LIN {X 0,Y 189.599,Z 448.711,A -85,B 0,C 180,E1 -22382.4,E2 -22382.4} C_VEL
LIN {X 0,Y 185.907,Z 453.993,A -85,B 0,C 180,E1 -22385.43,E2 -22385.43} C_VEL
LIN {X 0,Y 182.746,Z 458.185,A -85,B 0,C 180,E1 -22388.573,E2 -22388.573} C_VEL
LIN {X 0,Y 180.103,Z 461.393,A -85,B 0,C 180,E1 -22391.811,E2 -22391.811} C_VEL
LIN {X 0,Y 178.683,Z 463.032,A -85,B 0,C 180,E1 -22394.02,E2 -22394.02} C_VEL
LIN {X 0,Y 176.938,Z 465.065,A -85,B 0,C 180,E1 -22398.546,E2 -22398.546} C_VEL
LIN {X 0,Y 176.13,Z 465.589,A -85,B 0,C 180,E1 -22403.125,E2 -22403.125} C_VEL
LIN {X 0,Y 176.1,Z 465.056,A -85,B 0,C 180,E1 -22406.147,E2 -22406.147} C_VEL
LIN {X 0,Y 176.317,Z 464.526,A -85,B 0,C 180,E1 -22407.716,E2 -22407.716} C_VEL
LIN {X 0,Y 176.425,Z 463.36,A -85,B 0,C 180,E1 -22410,E2 -22410} C_VEL
LIN {X 0,Y 176.412,Z 461.752,A -85,B 0,C 180,E1 -22412.283,E2 -22412.283} C_VEL
LIN {X 0,Y 176.345,Z 458.528,A -85,B 0,C 180,E1 -22415.603,E2 -22415.603} C_VEL
LIN {X 0,Y 176.58,Z 453.896,A -85,B 0,C 180,E1 -22419.159,E2 -22419.159} C_VEL
LIN {X 0,Y 177.26,Z 448.101,A -85,B 0,C 180,E1 -22422.594,E2 -22422.594} C_VEL
LIN {X 0,Y 178.483,Z 440.77,A -85,B 0,C 180,E1 -22425.998,E2 -22425.998} C_VEL
LIN {X 0,Y 179.896,Z 433.284,A -85,B 0,C 180,E1 -22428.8,E2 -22428.8} C_VEL
LIN {X 0,Y 181.89,Z 423.485,A -85,B 0,C 180,E1 -22431.754,E2 -22431.754} C_VEL
LIN {X 0,Y 183.937,Z 412.997,A -85,B 0,C 180,E1 -22434.248,E2 -22434.248} C_VEL
LIN {X 0,Y 186.015,Z 401.711,A -85,B 0,C 180,E1 -22436.352,E2 -22436.352} C_VEL
LIN {X 0,Y 188.191,Z 389.227,A -85,B 0,C 180,E1 -22438.127,E2 -22438.127} C_VEL
LIN {X 0,Y 189.916,Z 375.866,A -85,B 0,C 180,E1 -22439.51,E2 -22439.51} C_VEL
LIN {X 0,Y 191.178,Z 362.832,A -85,B 0,C 180,E1 -22440.435,E2 -22440.435} C_VEL
LIN {X 0,Y 193.662,Z 313.849,A -85,B 0,C 180,E1 -22442.625,E2 -22442.625} C_VEL
LIN {X 0,Y 190.578,Z 284.083,A -85,B 0,C 180,E1 -22444.515,E2 -22444.515} C_VEL
LIN {X 0,Y 182.555,Z 261.017,A -85,B 0,C 180,E1 -22446.816,E2 -22446.816} C_VEL
LIN {X 0,Y 180.086,Z 254.3,A -85,B 0,C 180,E1 -22447.559,E2 -22447.559} C_VEL
LIN {X 0,Y 178.442,Z 247.259,A -85,B 0,C 180,E1 -22451.351,E2 -22451.351} C_VEL
LIN {X 0,Y 178.382,Z 247.27,A -85,B 0,C 180,E1 -22455.161,E2 -22455.161} C_VEL
LIN {X 0,Y 178.388,Z 247.265,A -85,B 0,C 180,E1 -22458.457,E2 -22458.457} C_VEL
LIN {X 0,Y 178.406,Z 247.261,A -85,B 0,C 180,E1 -22463.778,E2 -22463.778} C_VEL
LIN {X 0,Y 178.468,Z 247.249,A -85,B 0,C 180,E1 -22466.542,E2 -22466.542} C_VEL
LIN {X 0,Y 178.434,Z 247.254,A -85,B 0,C 180,E1 -22471.793,E2 -22471.793} C_VEL
LIN {X 0,Y 178.5,Z 247.242,A -85,B 0,C 180,E1 -22474.886,E2 -22474.886} C_VEL
LIN {X 0,Y 178.587,Z 247.231,A -85,B 0,C 180,E1 -22481.649,E2 -22481.649} C_VEL
LIN {X 0,Y 178.618,Z 247.225,A -85,B 0,C 180,E1 -22486.344,E2 -22486.344} C_VEL
LIN {X 0,Y 178.883,Z 247.204,A -85,B 0,C 180,E1 -22490.958,E2 -22490.958} C_VEL
LIN {X 0,Y 179.11,Z 247.151,A -85,B 0,C 180,E1 -22497.75,E2 -22497.75} C_VEL
LIN {X 0,Y 179.333,Z 247.119,A -85,B 0,C 180,E1 -22499.999,E2 -22499.999} C_VEL
LIN {X 0,Y 178.829,Z 247.202,A -85,B 0,C 180,E1 -22504.507,E2 -22504.507} C_VEL
LIN {X 0,Y 178.883,Z 247.202,A -85,B 0,C 180,E1 -22509.041,E2 -22509.041} C_VEL
LIN {X 0,Y 178.629,Z 247.222,A -85,B 0,C 180,E1 -22513.654,E2 -22513.654} C_VEL
LIN {X 0,Y 178.635,Z 247.195,A -85,B 0,C 180,E1 -22519.245,E2 -22519.245} C_VEL
LIN {X 0,Y 178.517,Z 247.242,A -85,B 0,C 180,E1 -22525.126,E2 -22525.126} C_VEL
LIN {X 0,Y 178.505,Z 247.249,A -85,B 0,C 180,E1 -22529.995,E2 -22529.995} C_VEL
LIN {X 0,Y 178.474,Z 247.243,A -85,B 0,C 180,E1 -22534.224,E2 -22534.224} C_VEL
LIN {X 0,Y 178.431,Z 247.223,A -85,B 0,C 180,E1 -22539.064,E2 -22539.064} C_VEL
LIN {X 0,Y 178.432,Z 247.234,A -85,B 0,C 180,E1 -22542.034,E2 -22542.034} C_VEL
LIN {X 0,Y 178.414,Z 247.253,A -85,B 0,C 180,E1 -22545.156,E2 -22545.156} C_VEL
LIN {X 0,Y 178.397,Z 247.263,A -85,B 0,C 180,E1 -22548.46,E2 -22548.46} C_VEL
LIN {X 0,Y 178.412,Z 247.252,A -85,B 0,C 180,E1 -22553.786,E2 -22553.786} C_VEL
LIN {X 0,Y 178.477,Z 247.23,A -85,B 0,C 180,E1 -22556.549,E2 -22556.549} C_VEL
LIN {X 0,Y 178.515,Z 247.234,A -85,B 0,C 180,E1 -22560.01,E2 -22560.01} C_VEL
LIN {X 0,Y 178.529,Z 247.246,A -85,B 0,C 180,E1 -22564.878,E2 -22564.878} C_VEL
LIN {X 0,Y 178.619,Z 247.221,A -85,B 0,C 180,E1 -22570.786,E2 -22570.786} C_VEL
LIN {X 0,Y 178.662,Z 247.228,A -85,B 0,C 180,E1 -22574.019,E2 -22574.019} C_VEL
LIN {X 0,Y 178.859,Z 247.2,A -85,B 0,C 180,E1 -22579.211,E2 -22579.211} C_VEL
LIN {X 0,Y 178.923,Z 247.198,A -85,B 0,C 180,E1 -22583.234,E2 -22583.234} C_VEL
LIN {X 0,Y 179.152,Z 247.165,A -85,B 0,C 180,E1 -22587.752,E2 -22587.752} C_VEL
LIN {X 0,Y 179.369,Z 247.142,A -85,B 0,C 180,E1 -22590,E2 -22590} C_VEL
LIN {X 0,Y 178.869,Z 247.204,A -85,B 0,C 180,E1 -22594.507,E2 -22594.507} C_VEL
LIN {X 0,Y 178.922,Z 247.2,A -85,B 0,C 180,E1 -22599.039,E2 -22599.039} C_VEL
LIN {X 0,Y 178.707,Z 247.228,A -85,B 0,C 180,E1 -22602.793,E2 -22602.793} C_VEL
LIN {X 0,Y 179.772,Z 250.154,A -85,B 0,C 180,E1 -22603.121,E2 -22603.121} C_VEL
LIN {X 0,Y 187.477,Z 267.491,A -85,B 0,C 180,E1 -22605.177,E2 -22605.177} C_VEL
LIN {X 0,Y 194.565,Z 285.188,A -85,B 0,C 180,E1 -22606.986,E2 -22606.986} C_VEL
LIN {X 0,Y 194.878,Z 286.201,A -85,B 0,C 180,E1 -22607.076,E2 -22607.076} C_VEL
LIN {X 0,Y 191.309,Z 347.18,A -85,B 0,C 180,E1 -22609.758,E2 -22609.758} C_VEL
LIN {X 0,Y 190.227,Z 360,A -85,B 0,C 180,E1 -22610.722,E2 -22610.722} C_VEL
LIN {X 0,Y 188.85,Z 371.973,A -85,B 0,C 180,E1 -22611.989,E2 -22611.989} C_VEL
LIN {X 0,Y 186.955,Z 384.854,A -85,B 0,C 180,E1 -22613.833,E2 -22613.833} C_VEL
LIN {X 0,Y 184.919,Z 396.527,A -85,B 0,C 180,E1 -22616.003,E2 -22616.003} C_VEL
LIN {X 0,Y 182.877,Z 407.104,A -85,B 0,C 180,E1 -22618.514,E2 -22618.514} C_VEL
LIN {X 0,Y 181.019,Z 416.582,A -85,B 0,C 180,E1 -22621.337,E2 -22621.337} C_VEL
LIN {X 0,Y 179.188,Z 425.253,A -85,B 0,C 180,E1 -22624.55,E2 -22624.55} C_VEL
LIN {X 0,Y 177.846,Z 432.169,A -85,B 0,C 180,E1 -22627.783,E2 -22627.783} C_VEL
LIN {X 0,Y 176.977,Z 437.712,A -85,B 0,C 180,E1 -22631.018,E2 -22631.018} C_VEL
LIN {X 0,Y 176.14,Z 443.11,A -85,B 0,C 180,E1 -22635.12,E2 -22635.12} C_VEL
LIN {X 0,Y 175.887,Z 445.264,A -85,B 0,C 180,E1 -22637.214,E2 -22637.214} C_VEL
LIN {X 0,Y 175.78,Z 447.658,A -85,B 0,C 180,E1 -22640.231,E2 -22640.231} C_VEL
LIN {X 0,Y 175.992,Z 449.322,A -85,B 0,C 180,E1 -22643.202,E2 -22643.202} C_VEL
LIN {X 0,Y 176.702,Z 450.396,A -85,B 0,C 180,E1 -22646.631,E2 -22646.631} C_VEL
LIN {X 0,Y 177.97,Z 450.542,A -85,B 0,C 180,E1 -22650.306,E2 -22650.306} C_VEL
LIN {X 0,Y 180.201,Z 449.345,A -85,B 0,C 180,E1 -22654.596,E2 -22654.596} C_VEL
LIN {X 0,Y 182.337,Z 447.564,A -85,B 0,C 180,E1 -22657.662,E2 -22657.662} C_VEL
LIN {X 0,Y 185.512,Z 444.303,A -85,B 0,C 180,E1 -22661.264,E2 -22661.264} C_VEL
LIN {X 0,Y 189.738,Z 439.371,A -85,B 0,C 180,E1 -22664.973,E2 -22664.973} C_VEL
LIN {X 0,Y 193.955,Z 433.791,A -85,B 0,C 180,E1 -22668.027,E2 -22668.027} C_VEL
LIN {X 0,Y 197.968,Z 427.738,A -85,B 0,C 180,E1 -22670.602,E2 -22670.602} C_VEL
LIN {X 0,Y 202.399,Z 420.472,A -85,B 0,C 180,E1 -22673.02,E2 -22673.02} C_VEL
LIN {X 0,Y 207.339,Z 411.368,A -85,B 0,C 180,E1 -22675.383,E2 -22675.383} C_VEL
LIN {X 0,Y 212.434,Z 400.451,A -85,B 0,C 180,E1 -22677.574,E2 -22677.574} C_VEL
LIN {X 0,Y 216.736,Z 389.318,A -85,B 0,C 180,E1 -22679.289,E2 -22679.289} C_VEL
LIN {X 0,Y 220.567,Z 377.326,A -85,B 0,C 180,E1 -22680.685,E2 -22680.685} C_VEL
LIN {X 0,Y 223.601,Z 364.833,A -85,B 0,C 180,E1 -22681.802,E2 -22681.802} C_VEL
LIN {X 0,Y 225.801,Z 352.533,A -85,B 0,C 180,E1 -22682.584,E2 -22682.584} C_VEL
LIN {X 0,Y 228.467,Z 329.492,A -85,B 0,C 180,E1 -22683.486,E2 -22683.486} C_VEL
LIN {X 0,Y 230.182,Z 313.067,A -85,B 0,C 180,E1 -22684.103,E2 -22684.103} C_VEL
LIN {X 0,Y 226.331,Z 304.592,A -85,B 0,C 180,E1 -22686.72,E2 -22686.72} C_VEL
LIN {X 0,Y 224.187,Z 300.987,A -85,B 0,C 180,E1 -22688.303,E2 -22688.303} C_VEL
LIN {X 0,Y 221.023,Z 295.846,A -85,B 0,C 180,E1 -22690.999,E2 -22690.999} C_VEL
LIN {X 0,Y 219.416,Z 293.216,A -85,B 0,C 180,E1 -22692.625,E2 -22692.625} C_VEL
LIN {X 0,Y 217.287,Z 290.254,A -85,B 0,C 180,E1 -22695.197,E2 -22695.197} C_VEL
LIN {X 0,Y 215.463,Z 287.989,A -85,B 0,C 180,E1 -22698.105,E2 -22698.105} C_VEL
LIN {X 0,Y 214.273,Z 286.482,A -85,B 0,C 180,E1 -22701.15,E2 -22701.15} C_VEL
LIN {X 0,Y 213.854,Z 286.773,A -85,B 0,C 180,E1 -22706.485,E2 -22706.485} C_VEL
LIN {X 0,Y 214.9,Z 288.985,A -85,B 0,C 180,E1 -22710.453,E2 -22710.453} C_VEL
LIN {X 0,Y 217.907,Z 295.087,A -85,B 0,C 180,E1 -22715.571,E2 -22715.571} C_VEL
LIN {X 0,Y 220.497,Z 300.345,A -85,B 0,C 180,E1 -22718.445,E2 -22718.445} C_VEL
LIN {X 0,Y 223.12,Z 306.049,A -85,B 0,C 180,E1 -22720.845,E2 -22720.845} C_VEL
LIN {X 0,Y 225.734,Z 312.199,A -85,B 0,C 180,E1 -22722.959,E2 -22722.959} C_VEL
LIN {X 0,Y 228.58,Z 319.942,A -85,B 0,C 180,E1 -22725.006,E2 -22725.006} C_VEL
LIN {X 0,Y 229.366,Z 322.663,A -85,B 0,C 180,E1 -22725.588,E2 -22725.588} C_VEL
LIN {X 0,Y 229.11,Z 326.685,A -85,B 0,C 180,E1 -22725.81,E2 -22725.81} C_VEL
LIN {X 0,Y 225.297,Z 360.929,A -85,B 0,C 180,E1 -22727.075,E2 -22727.075} C_VEL
LIN {X 0,Y 224.524,Z 365.452,A -85,B 0,C 180,E1 -22727.265,E2 -22727.265} C_VEL
LIN {X 0,Y 223.429,Z 369.295,A -85,B 0,C 180,E1 -22727.323,E2 -22727.323} C_VEL
LIN {X 0,Y 217.491,Z 381.326,A -85,B 0,C 180,E1 -22726.845,E2 -22726.845} C_VEL
LIN {X 0,Y 216.118,Z 384.997,A -85,B 0,C 180,E1 -22727.019,E2 -22727.019} C_VEL
LIN {X 0,Y 212.124,Z 396.806,A -85,B 0,C 180,E1 -22728.187,E2 -22728.187} C_VEL
LIN {X 0,Y 207.021,Z 409.179,A -85,B 0,C 180,E1 -22729.838,E2 -22729.838} C_VEL
LIN {X 0,Y 201.733,Z 420.185,A -85,B 0,C 180,E1 -22731.807,E2 -22731.807} C_VEL
LIN {X 0,Y 196.789,Z 429.15,A -85,B 0,C 180,E1 -22733.899,E2 -22733.899} C_VEL
LIN {X 0,Y 191.316,Z 437.995,A -85,B 0,C 180,E1 -22736.567,E2 -22736.567} C_VEL
LIN {X 0,Y 186.364,Z 445.214,A -85,B 0,C 180,E1 -22739.4,E2 -22739.4} C_VEL
LIN {X 0,Y 181.983,Z 451.123,A -85,B 0,C 180,E1 -22742.395,E2 -22742.395} C_VEL
LIN {X 0,Y 178.293,Z 455.843,A -85,B 0,C 180,E1 -22745.553,E2 -22745.553} C_VEL
LIN {X 0,Y 175.164,Z 459.516,A -85,B 0,C 180,E1 -22748.834,E2 -22748.834} C_VEL
LIN {X 0,Y 173.364,Z 461.453,A -85,B 0,C 180,E1 -22751.078,E2 -22751.078} C_VEL
LIN {X 0,Y 170.739,Z 464.082,A -85,B 0,C 180,E1 -22755.703,E2 -22755.703} C_VEL
LIN {X 0,Y 169.386,Z 465.213,A -85,B 0,C 180,E1 -22760.448,E2 -22760.448} C_VEL
LIN {X 0,Y 169.082,Z 465.187,A -85,B 0,C 180,E1 -22762.837,E2 -22762.837} C_VEL
LIN {X 0,Y 169.242,Z 463.955,A -85,B 0,C 180,E1 -22767.62,E2 -22767.62} C_VEL
LIN {X 0,Y 169.364,Z 462.725,A -85,B 0,C 180,E1 -22770,E2 -22770} C_VEL
LIN {X 0,Y 169.269,Z 459.946,A -85,B 0,C 180,E1 -22773.591,E2 -22773.591} C_VEL
LIN {X 0,Y 169.327,Z 456.088,A -85,B 0,C 180,E1 -22777.152,E2 -22777.152} C_VEL
LIN {X 0,Y 169.771,Z 451,A -85,B 0,C 180,E1 -22780.735,E2 -22780.735} C_VEL
LIN {X 0,Y 170.659,Z 444.517,A -85,B 0,C 180,E1 -22784.303,E2 -22784.303} C_VEL
LIN {X 0,Y 172.216,Z 436.375,A -85,B 0,C 180,E1 -22787.82,E2 -22787.82} C_VEL
LIN {X 0,Y 173.845,Z 428.029,A -85,B 0,C 180,E1 -22790.713,E2 -22790.713} C_VEL
LIN {X 0,Y 175.971,Z 417.858,A -85,B 0,C 180,E1 -22793.537,E2 -22793.537} C_VEL
LIN {X 0,Y 178.275,Z 406.408,A -85,B 0,C 180,E1 -22796.01,E2 -22796.01} C_VEL
LIN {X 0,Y 180.296,Z 395.287,A -85,B 0,C 180,E1 -22797.886,E2 -22797.886} C_VEL
LIN {X 0,Y 182.206,Z 383.022,A -85,B 0,C 180,E1 -22799.454,E2 -22799.454} C_VEL
LIN {X 0,Y 183.801,Z 369.682,A -85,B 0,C 180,E1 -22800.675,E2 -22800.675} C_VEL
LIN {X 0,Y 184.836,Z 356.969,A -85,B 0,C 180,E1 -22801.437,E2 -22801.437} C_VEL
LIN {X 0,Y 187.018,Z 314.116,A -85,B 0,C 180,E1 -22803.404,E2 -22803.404} C_VEL
LIN {X 0,Y 184.2,Z 286.195,A -85,B 0,C 180,E1 -22805.224,E2 -22805.224} C_VEL
LIN {X 0,Y 176.567,Z 264.085,A -85,B 0,C 180,E1 -22807.542,E2 -22807.542} C_VEL
LIN {X 0,Y 172.741,Z 253.927,A -85,B 0,C 180,E1 -22808.734,E2 -22808.734} C_VEL
LIN {X 0,Y 171.377,Z 248.14,A -85,B 0,C 180,E1 -22812,E2 -22812} C_VEL
LIN {X 0,Y 171.322,Z 248.148,A -85,B 0,C 180,E1 -22817.588,E2 -22817.588} C_VEL
LIN {X 0,Y 171.348,Z 248.142,A -85,B 0,C 180,E1 -22822.03,E2 -22822.03} C_VEL
LIN {X 0,Y 171.385,Z 248.132,A -85,B 0,C 180,E1 -22825.09,E2 -22825.09} C_VEL
LIN {X 0,Y 171.397,Z 248.135,A -85,B 0,C 180,E1 -22830.524,E2 -22830.524} C_VEL
LIN {X 0,Y 171.419,Z 248.129,A -85,B 0,C 180,E1 -22835.795,E2 -22835.795} C_VEL
LIN {X 0,Y 171.488,Z 248.12,A -85,B 0,C 180,E1 -22840.86,E2 -22840.86} C_VEL
LIN {X 0,Y 171.533,Z 248.105,A -85,B 0,C 180,E1 -22845.768,E2 -22845.768} C_VEL
LIN {X 0,Y 171.822,Z 248.082,A -85,B 0,C 180,E1 -22850.583,E2 -22850.583} C_VEL
LIN {X 0,Y 171.774,Z 248.076,A -85,B 0,C 180,E1 -22855.305,E2 -22855.305} C_VEL
LIN {X 0,Y 172.297,Z 247.994,A -85,B 0,C 180,E1 -22859.999,E2 -22859.999} C_VEL
LIN {X 0,Y 171.778,Z 248.081,A -85,B 0,C 180,E1 -22864.693,E2 -22864.693} C_VEL
LIN {X 0,Y 171.822,Z 248.08,A -85,B 0,C 180,E1 -22869.416,E2 -22869.416} C_VEL
LIN {X 0,Y 171.549,Z 248.1,A -85,B 0,C 180,E1 -22874.229,E2 -22874.229} C_VEL
LIN {X 0,Y 171.557,Z 248.077,A -85,B 0,C 180,E1 -22879.591,E2 -22879.591} C_VEL
LIN {X 0,Y 171.452,Z 248.121,A -85,B 0,C 180,E1 -22885.617,E2 -22885.617} C_VEL
LIN {X 0,Y 171.423,Z 248.131,A -85,B 0,C 180,E1 -22890.587,E2 -22890.587} C_VEL
LIN {X 0,Y 171.386,Z 248.122,A -85,B 0,C 180,E1 -22895.035,E2 -22895.035} C_VEL
LIN {X 0,Y 171.387,Z 248.099,A -85,B 0,C 180,E1 -22898.828,E2 -22898.828} C_VEL
LIN {X 0,Y 171.342,Z 248.129,A -85,B 0,C 180,E1 -22904.209,E2 -22904.209} C_VEL
LIN {X 0,Y 171.328,Z 248.142,A -85,B 0,C 180,E1 -22908.985,E2 -22908.985} C_VEL
LIN {X 0,Y 171.376,Z 248.134,A -85,B 0,C 180,E1 -22912.043,E2 -22912.043} C_VEL
LIN {X 0,Y 171.389,Z 248.121,A -85,B 0,C 180,E1 -22915.095,E2 -22915.095} C_VEL
LIN {X 0,Y 171.442,Z 248.119,A -85,B 0,C 180,E1 -22920.537,E2 -22920.537} C_VEL
LIN {X 0,Y 171.453,Z 248.129,A -85,B 0,C 180,E1 -22925.804,E2 -22925.804} C_VEL
LIN {X 0,Y 171.575,Z 248.097,A -85,B 0,C 180,E1 -22930.874,E2 -22930.874} C_VEL
LIN {X 0,Y 171.607,Z 248.11,A -85,B 0,C 180,E1 -22935.777,E2 -22935.777} C_VEL
LIN {X 0,Y 171.871,Z 248.065,A -85,B 0,C 180,E1 -22940.587,E2 -22940.587} C_VEL
LIN {X 0,Y 171.821,Z 248.084,A -85,B 0,C 180,E1 -22945.308,E2 -22945.308} C_VEL
LIN {X 0,Y 172.332,Z 248.019,A -85,B 0,C 180,E1 -22950,E2 -22950} C_VEL
LIN {X 0,Y 171.818,Z 248.083,A -85,B 0,C 180,E1 -22954.692,E2 -22954.692} C_VEL
LIN {X 0,Y 171.86,Z 248.079,A -85,B 0,C 180,E1 -22959.414,E2 -22959.414} C_VEL
LIN {X 0,Y 171.734,Z 248.097,A -85,B 0,C 180,E1 -22961.7,E2 -22961.7} C_VEL
LIN {X 0,Y 172.764,Z 251.05,A -85,B 0,C 180,E1 -22962.069,E2 -22962.069} C_VEL
LIN {X 0,Y 180.588,Z 268.538,A -85,B 0,C 180,E1 -22964.262,E2 -22964.262} C_VEL
LIN {X 0,Y 188.151,Z 287.318,A -85,B 0,C 180,E1 -22966.296,E2 -22966.296} C_VEL
LIN {X 0,Y 184.635,Z 347.103,A -85,B 0,C 180,E1 -22969.032,E2 -22969.032} C_VEL
LIN {X 0,Y 183.493,Z 360.308,A -85,B 0,C 180,E1 -22970.053,E2 -22970.053} C_VEL
LIN {X 0,Y 182.053,Z 372.503,A -85,B 0,C 180,E1 -22971.391,E2 -22971.391} C_VEL
LIN {X 0,Y 180.105,Z 385.172,A -85,B 0,C 180,E1 -22973.269,E2 -22973.269} C_VEL
LIN {X 0,Y 177.949,Z 397.03,A -85,B 0,C 180,E1 -22975.553,E2 -22975.553} C_VEL
LIN {X 0,Y 175.828,Z 407.778,A -85,B 0,C 180,E1 -22978.219,E2 -22978.219} C_VEL
LIN {X 0,Y 173.75,Z 417.822,A -85,B 0,C 180,E1 -22981.359,E2 -22981.359} C_VEL
LIN {X 0,Y 171.872,Z 426.748,A -85,B 0,C 180,E1 -22984.919,E2 -22984.919} C_VEL
LIN {X 0,Y 170.5,Z 433.74,A -85,B 0,C 180,E1 -22988.449,E2 -22988.449} C_VEL
LIN {X 0,Y 169.676,Z 439.007,A -85,B 0,C 180,E1 -22991.794,E2 -22991.794} C_VEL
LIN {X 0,Y 169.046,Z 443.038,A -85,B 0,C 180,E1 -22995.029,E2 -22995.029} C_VEL
LIN {X 0,Y 168.689,Z 446.419,A -85,B 0,C 180,E1 -22998.577,E2 -22998.577} C_VEL
LIN {X 0,Y 168.802,Z 448.905,A -85,B 0,C 180,E1 -23002.277,E2 -23002.277} C_VEL
LIN {X 0,Y 169.436,Z 450.426,A -85,B 0,C 180,E1 -23006.046,E2 -23006.046} C_VEL
LIN {X 0,Y 170.875,Z 450.942,A -85,B 0,C 180,E1 -23010.427,E2 -23010.427} C_VEL
LIN {X 0,Y 172.462,Z 450.43,A -85,B 0,C 180,E1 -23013.692,E2 -23013.692} C_VEL
LIN {X 0,Y 174.948,Z 448.818,A -85,B 0,C 180,E1 -23017.497,E2 -23017.497} C_VEL
LIN {X 0,Y 178.538,Z 445.664,A -85,B 0,C 180,E1 -23021.645,E2 -23021.645} C_VEL
LIN {X 0,Y 183.291,Z 440.631,A -85,B 0,C 180,E1 -23025.805,E2 -23025.805} C_VEL
LIN {X 0,Y 188.158,Z 434.69,A -85,B 0,C 180,E1 -23029.237,E2 -23029.237} C_VEL
LIN {X 0,Y 192.925,Z 428.065,A -85,B 0,C 180,E1 -23032.149,E2 -23032.149} C_VEL
LIN {X 0,Y 198.15,Z 419.954,A -85,B 0,C 180,E1 -23034.828,E2 -23034.828} C_VEL
LIN {X 0,Y 202.612,Z 412.123,A -85,B 0,C 180,E1 -23036.854,E2 -23036.854} C_VEL
LIN {X 0,Y 207.866,Z 401.396,A -85,B 0,C 180,E1 -23039.032,E2 -23039.032} C_VEL
LIN {X 0,Y 212.257,Z 390.85,A -85,B 0,C 180,E1 -23040.697,E2 -23040.697} C_VEL
LIN {X 0,Y 216.042,Z 379.905,A -85,B 0,C 180,E1 -23042.022,E2 -23042.022} C_VEL
LIN {X 0,Y 219.409,Z 367.366,A -85,B 0,C 180,E1 -23043.204,E2 -23043.204} C_VEL
LIN {X 0,Y 221.991,Z 354.424,A -85,B 0,C 180,E1 -23044.061,E2 -23044.061} C_VEL
LIN {X 0,Y 224.248,Z 336.519,A -85,B 0,C 180,E1 -23044.797,E2 -23044.797} C_VEL
LIN {X 0,Y 226.409,Z 316.645,A -85,B 0,C 180,E1 -23045.543,E2 -23045.543} C_VEL
LIN {X 0,Y 223.518,Z 309.761,A -85,B 0,C 180,E1 -23047.766,E2 -23047.766} C_VEL
LIN {X 0,Y 220.811,Z 305.409,A -85,B 0,C 180,E1 -23049.927,E2 -23049.927} C_VEL
LIN {X 0,Y 219.147,Z 302.331,A -85,B 0,C 180,E1 -23051.555,E2 -23051.555} C_VEL
LIN {X 0,Y 217.558,Z 299.751,A -85,B 0,C 180,E1 -23053.231,E2 -23053.231} C_VEL
LIN {X 0,Y 215.64,Z 296.775,A -85,B 0,C 180,E1 -23055.79,E2 -23055.79} C_VEL
LIN {X 0,Y 214.032,Z 294.763,A -85,B 0,C 180,E1 -23058.607,E2 -23058.607} C_VEL
LIN {X 0,Y 213.075,Z 293.462,A -85,B 0,C 180,E1 -23061.274,E2 -23061.274} C_VEL
LIN {X 0,Y 212.656,Z 293.737,A -85,B 0,C 180,E1 -23066.224,E2 -23066.224} C_VEL
LIN {X 0,Y 213.536,Z 295.748,A -85,B 0,C 180,E1 -23070.011,E2 -23070.011} C_VEL
LIN {X 0,Y 216.182,Z 301.608,A -85,B 0,C 180,E1 -23074.965,E2 -23074.965} C_VEL
LIN {X 0,Y 218.488,Z 306.657,A -85,B 0,C 180,E1 -23077.761,E2 -23077.761} C_VEL
LIN {X 0,Y 220.72,Z 311.934,A -85,B 0,C 180,E1 -23080.024,E2 -23080.024} C_VEL
LIN {X 0,Y 223.064,Z 317.744,A -85,B 0,C 180,E1 -23082.045,E2 -23082.045} C_VEL
LIN {X 0,Y 225.461,Z 324.846,A -85,B 0,C 180,E1 -23083.979,E2 -23083.979} C_VEL
LIN {X 0,Y 225.706,Z 326.211,A -85,B 0,C 180,E1 -23084.217,E2 -23084.217} C_VEL
LIN {X 0,Y 221.783,Z 360.31,A -85,B 0,C 180,E1 -23085.481,E2 -23085.481} C_VEL
LIN {X 0,Y 219.295,Z 373.01,A -85,B 0,C 180,E1 -23086.135,E2 -23086.135} C_VEL
LIN {X 0,Y 216.118,Z 384.997,A -85,B 0,C 180,E1 -23087.019,E2 -23087.019} C_VEL
LIN {X 0,Y 214.102,Z 390.411,A -85,B 0,C 180,E1 -23087.386,E2 -23087.386} C_VEL
LIN {X 0,Y 209.313,Z 399.052,A -85,B 0,C 180,E1 -23087.651,E2 -23087.651} C_VEL
LIN {X 0,Y 204.132,Z 407.359,A -85,B 0,C 180,E1 -23088.068,E2 -23088.068} C_VEL
LIN {X 0,Y 201.518,Z 412.109,A -85,B 0,C 180,E1 -23088.685,E2 -23088.685} C_VEL
LIN {X 0,Y 197.401,Z 420,A -85,B 0,C 180,E1 -23090.15,E2 -23090.15} C_VEL
LIN {X 0,Y 191.188,Z 430.505,A -85,B 0,C 180,E1 -23092.665,E2 -23092.665} C_VEL
LIN {X 0,Y 185.496,Z 439.056,A -85,B 0,C 180,E1 -23095.371,E2 -23095.371} C_VEL
LIN {X 0,Y 180.338,Z 445.985,A -85,B 0,C 180,E1 -23098.261,E2 -23098.261} C_VEL
LIN {X 0,Y 174.835,Z 452.702,A -85,B 0,C 180,E1 -23102.025,E2 -23102.025} C_VEL
LIN {X 0,Y 170.672,Z 457.434,A -85,B 0,C 180,E1 -23105.686,E2 -23105.686} C_VEL
LIN {X 0,Y 168.538,Z 459.673,A -85,B 0,C 180,E1 -23107.96,E2 -23107.96} C_VEL
LIN {X 0,Y 165.046,Z 462.892,A -85,B 0,C 180,E1 -23112.66,E2 -23112.66} C_VEL
LIN {X 0,Y 162.978,Z 464.601,A -85,B 0,C 180,E1 -23117.55,E2 -23117.55} C_VEL
LIN {X 0,Y 162.017,Z 464.737,A -85,B 0,C 180,E1 -23122.523,E2 -23122.523} C_VEL
LIN {X 0,Y 162.165,Z 463.36,A -85,B 0,C 180,E1 -23127.516,E2 -23127.516} C_VEL
LIN {X 0,Y 162.304,Z 462.043,A -85,B 0,C 180,E1 -23130,E2 -23130} C_VEL
LIN {X 0,Y 162.21,Z 459.366,A -85,B 0,C 180,E1 -23133.487,E2 -23133.487} C_VEL
LIN {X 0,Y 162.267,Z 455.127,A -85,B 0,C 180,E1 -23137.465,E2 -23137.465} C_VEL
LIN {X 0,Y 162.898,Z 448.826,A -85,B 0,C 180,E1 -23141.824,E2 -23141.824} C_VEL
LIN {X 0,Y 164.014,Z 441.888,A -85,B 0,C 180,E1 -23145.532,E2 -23145.532} C_VEL
LIN {X 0,Y 165.41,Z 434.777,A -85,B 0,C 180,E1 -23148.58,E2 -23148.58} C_VEL
LIN {X 0,Y 167.192,Z 426.173,A -85,B 0,C 180,E1 -23151.578,E2 -23151.578} C_VEL
LIN {X 0,Y 169.427,Z 415.551,A -85,B 0,C 180,E1 -23154.504,E2 -23154.504} C_VEL
LIN {X 0,Y 171.586,Z 405.117,A -85,B 0,C 180,E1 -23156.775,E2 -23156.775} C_VEL
LIN {X 0,Y 173.723,Z 393.768,A -85,B 0,C 180,E1 -23158.708,E2 -23158.708} C_VEL
LIN {X 0,Y 175.694,Z 381.042,A -85,B 0,C 180,E1 -23160.329,E2 -23160.329} C_VEL
LIN {X 0,Y 177.274,Z 367.984,A -85,B 0,C 180,E1 -23161.517,E2 -23161.517} C_VEL
LIN {X 0,Y 178.305,Z 354.272,A -85,B 0,C 180,E1 -23162.311,E2 -23162.311} C_VEL
LIN {X 0,Y 180.374,Z 314.424,A -85,B 0,C 180,E1 -23164.209,E2 -23164.209} C_VEL
LIN {X 0,Y 177.684,Z 287.859,A -85,B 0,C 180,E1 -23166.035,E2 -23166.035} C_VEL
LIN {X 0,Y 170.641,Z 267.261,A -85,B 0,C 180,E1 -23168.287,E2 -23168.287} C_VEL
LIN {X 0,Y 165.369,Z 253.581,A -85,B 0,C 180,E1 -23170.011,E2 -23170.011} C_VEL
LIN {X 0,Y 164.288,Z 249.025,A -85,B 0,C 180,E1 -23172.738,E2 -23172.738} C_VEL
LIN {X 0,Y 164.251,Z 249.03,A -85,B 0,C 180,E1 -23176.794,E2 -23176.794} C_VEL
LIN {X 0,Y 164.279,Z 249.022,A -85,B 0,C 180,E1 -23180.351,E2 -23180.351} C_VEL
LIN {X 0,Y 164.313,Z 249.014,A -85,B 0,C 180,E1 -23184.348,E2 -23184.348} C_VEL
LIN {X 0,Y 164.357,Z 249.013,A -85,B 0,C 180,E1 -23189.127,E2 -23189.127} C_VEL
LIN {X 0,Y 164.38,Z 249,A -85,B 0,C 180,E1 -23194.687,E2 -23194.687} C_VEL
LIN {X 0,Y 164.4,Z 249.004,A -85,B 0,C 180,E1 -23200.115,E2 -23200.115} C_VEL
LIN {X 0,Y 164.461,Z 248.98,A -85,B 0,C 180,E1 -23205.142,E2 -23205.142} C_VEL
LIN {X 0,Y 164.744,Z 248.963,A -85,B 0,C 180,E1 -23210.174,E2 -23210.174} C_VEL
LIN {X 0,Y 164.8,Z 248.956,A -85,B 0,C 180,E1 -23212.649,E2 -23212.649} C_VEL
LIN {X 0,Y 165.261,Z 248.869,A -85,B 0,C 180,E1 -23219.999,E2 -23219.999} C_VEL
LIN {X 0,Y 164.727,Z 248.96,A -85,B 0,C 180,E1 -23224.894,E2 -23224.894} C_VEL
LIN {X 0,Y 164.801,Z 248.956,A -85,B 0,C 180,E1 -23227.349,E2 -23227.349} C_VEL
LIN {X 0,Y 164.682,Z 248.966,A -85,B 0,C 180,E1 -23231.056,E2 -23231.056} C_VEL
LIN {X 0,Y 164.478,Z 248.958,A -85,B 0,C 180,E1 -23237.403,E2 -23237.403} C_VEL
LIN {X 0,Y 164.486,Z 248.958,A -85,B 0,C 180,E1 -23239.987,E2 -23239.987} C_VEL
LIN {X 0,Y 164.376,Z 249.004,A -85,B 0,C 180,E1 -23246.135,E2 -23246.135} C_VEL
LIN {X 0,Y 164.358,Z 249.009,A -85,B 0,C 180,E1 -23251.228,E2 -23251.228} C_VEL
LIN {X 0,Y 164.301,Z 248.994,A -85,B 0,C 180,E1 -23256.787,E2 -23256.787} C_VEL
LIN {X 0,Y 164.302,Z 248.979,A -85,B 0,C 180,E1 -23259.912,E2 -23259.912} C_VEL
LIN {X 0,Y 164.295,Z 249.002,A -85,B 0,C 180,E1 -23263.355,E2 -23263.355} C_VEL
LIN {X 0,Y 164.282,Z 249.018,A -85,B 0,C 180,E1 -23266.811,E2 -23266.811} C_VEL
LIN {X 0,Y 164.286,Z 249.02,A -85,B 0,C 180,E1 -23270.355,E2 -23270.355} C_VEL
LIN {X 0,Y 164.321,Z 249.003,A -85,B 0,C 180,E1 -23274.352,E2 -23274.352} C_VEL
LIN {X 0,Y 164.382,Z 248.988,A -85,B 0,C 180,E1 -23279.137,E2 -23279.137} C_VEL
LIN {X 0,Y 164.411,Z 249.005,A -85,B 0,C 180,E1 -23284.696,E2 -23284.696} C_VEL
LIN {X 0,Y 164.481,Z 248.982,A -85,B 0,C 180,E1 -23290.053,E2 -23290.053} C_VEL
LIN {X 0,Y 164.55,Z 248.986,A -85,B 0,C 180,E1 -23295.154,E2 -23295.154} C_VEL
LIN {X 0,Y 164.795,Z 248.947,A -85,B 0,C 180,E1 -23300.179,E2 -23300.179} C_VEL
LIN {X 0,Y 164.845,Z 248.949,A -85,B 0,C 180,E1 -23302.653,E2 -23302.653} C_VEL
LIN {X 0,Y 165.048,Z 248.921,A -85,B 0,C 180,E1 -23307.56,E2 -23307.56} C_VEL
LIN {X 0,Y 165.294,Z 248.896,A -85,B 0,C 180,E1 -23310,E2 -23310} C_VEL
LIN {X 0,Y 164.767,Z 248.962,A -85,B 0,C 180,E1 -23314.893,E2 -23314.893} C_VEL
LIN {X 0,Y 164.836,Z 248.953,A -85,B 0,C 180,E1 -23317.348,E2 -23317.348} C_VEL
LIN {X 0,Y 164.765,Z 248.977,A -85,B 0,C 180,E1 -23320.584,E2 -23320.584} C_VEL
LIN {X 0,Y 165.755,Z 251.799,A -85,B 0,C 180,E1 -23320.935,E2 -23320.935} C_VEL
LIN {X 0,Y 174.683,Z 271.77,A -85,B 0,C 180,E1 -23323.559,E2 -23323.559} C_VEL
LIN {X 0,Y 181.563,Z 288.78,A -85,B 0,C 180,E1 -23325.504,E2 -23325.504} C_VEL
LIN {X 0,Y 177.982,Z 347.106,A -85,B 0,C 180,E1 -23328.255,E2 -23328.255} C_VEL
LIN {X 0,Y 176.802,Z 360.224,A -85,B 0,C 180,E1 -23329.293,E2 -23329.293} C_VEL
LIN {X 0,Y 175.313,Z 372.579,A -85,B 0,C 180,E1 -23330.686,E2 -23330.686} C_VEL
LIN {X 0,Y 173.377,Z 384.803,A -85,B 0,C 180,E1 -23332.539,E2 -23332.539} C_VEL
LIN {X 0,Y 171.341,Z 395.728,A -85,B 0,C 180,E1 -23334.673,E2 -23334.673} C_VEL
LIN {X 0,Y 169.323,Z 405.872,A -85,B 0,C 180,E1 -23337.163,E2 -23337.163} C_VEL
LIN {X 0,Y 167.478,Z 414.681,A -85,B 0,C 180,E1 -23339.843,E2 -23339.843} C_VEL
LIN {X 0,Y 165.724,Z 422.535,A -85,B 0,C 180,E1 -23342.772,E2 -23342.772} C_VEL
LIN {X 0,Y 164.165,Z 429.931,A -85,B 0,C 180,E1 -23346.185,E2 -23346.185} C_VEL
LIN {X 0,Y 162.897,Z 436.996,A -85,B 0,C 180,E1 -23350.322,E2 -23350.322} C_VEL
LIN {X 0,Y 162.116,Z 441.766,A -85,B 0,C 180,E1 -23353.912,E2 -23353.912} C_VEL
LIN {X 0,Y 161.672,Z 445.583,A -85,B 0,C 180,E1 -23357.64,E2 -23357.64} C_VEL
LIN {X 0,Y 161.732,Z 449.058,A -85,B 0,C 180,E1 -23362.53,E2 -23362.53} C_VEL
LIN {X 0,Y 162.238,Z 450.455,A -85,B 0,C 180,E1 -23365.727,E2 -23365.727} C_VEL
LIN {X 0,Y 163.302,Z 451.241,A -85,B 0,C 180,E1 -23369.389,E2 -23369.389} C_VEL
LIN {X 0,Y 165.09,Z 451.12,A -85,B 0,C 180,E1 -23373.366,E2 -23373.366} C_VEL
LIN {X 0,Y 167.984,Z 449.691,A -85,B 0,C 180,E1 -23377.882,E2 -23377.882} C_VEL
LIN {X 0,Y 170.749,Z 447.621,A -85,B 0,C 180,E1 -23381.186,E2 -23381.186} C_VEL
LIN {X 0,Y 174.677,Z 444.119,A -85,B 0,C 180,E1 -23384.91,E2 -23384.91} C_VEL
LIN {X 0,Y 179.723,Z 438.865,A -85,B 0,C 180,E1 -23388.726,E2 -23388.726} C_VEL
LIN {X 0,Y 184.58,Z 433.015,A -85,B 0,C 180,E1 -23391.833,E2 -23391.833} C_VEL
LIN {X 0,Y 189.242,Z 426.707,A -85,B 0,C 180,E1 -23394.41,E2 -23394.41} C_VEL
LIN {X 0,Y 194.465,Z 418.841,A -85,B 0,C 180,E1 -23396.894,E2 -23396.894} C_VEL
LIN {X 0,Y 200.102,Z 409.203,A -85,B 0,C 180,E1 -23399.246,E2 -23399.246} C_VEL
LIN {X 0,Y 205.236,Z 398.723,A -85,B 0,C 180,E1 -23401.211,E2 -23401.211} C_VEL
LIN {X 0,Y 210.037,Z 387.046,A -85,B 0,C 180,E1 -23402.887,E2 -23402.887} C_VEL
LIN {X 0,Y 214.134,Z 374.445,A -85,B 0,C 180,E1 -23404.236,E2 -23404.236} C_VEL
LIN {X 0,Y 217.122,Z 362.281,A -85,B 0,C 180,E1 -23405.224,E2 -23405.224} C_VEL
LIN {X 0,Y 219.361,Z 350.11,A -85,B 0,C 180,E1 -23405.898,E2 -23405.898} C_VEL
LIN {X 0,Y 222.88,Z 320.139,A -85,B 0,C 180,E1 -23407.056,E2 -23407.056} C_VEL
LIN {X 0,Y 220.851,Z 315.279,A -85,B 0,C 180,E1 -23408.758,E2 -23408.758} C_VEL
LIN {X 0,Y 217.217,Z 308.766,A -85,B 0,C 180,E1 -23412.188,E2 -23412.188} C_VEL
LIN {X 0,Y 215.868,Z 306.412,A -85,B 0,C 180,E1 -23413.752,E2 -23413.752} C_VEL
LIN {X 0,Y 213.76,Z 303.079,A -85,B 0,C 180,E1 -23416.762,E2 -23416.762} C_VEL
LIN {X 0,Y 212.021,Z 300.72,A -85,B 0,C 180,E1 -23420.676,E2 -23420.676} C_VEL
LIN {X 0,Y 211.458,Z 300.41,A -85,B 0,C 180,E1 -23423.506,E2 -23423.506} C_VEL
LIN {X 0,Y 211.532,Z 300.96,A -85,B 0,C 180,E1 -23426.783,E2 -23426.783} C_VEL
LIN {X 0,Y 212.236,Z 302.746,A -85,B 0,C 180,E1 -23429.783,E2 -23429.783} C_VEL
LIN {X 0,Y 214.512,Z 308.175,A -85,B 0,C 180,E1 -23434.391,E2 -23434.391} C_VEL
LIN {X 0,Y 216.564,Z 313.1,A -85,B 0,C 180,E1 -23437.133,E2 -23437.133} C_VEL
LIN {X 0,Y 218.557,Z 318.186,A -85,B 0,C 180,E1 -23439.332,E2 -23439.332} C_VEL
LIN {X 0,Y 220.789,Z 324.321,A -85,B 0,C 180,E1 -23441.425,E2 -23441.425} C_VEL
LIN {X 0,Y 222.152,Z 328.756,A -85,B 0,C 180,E1 -23442.659,E2 -23442.659} C_VEL
LIN {X 0,Y 218.314,Z 360.526,A -85,B 0,C 180,E1 -23443.872,E2 -23443.872} C_VEL
LIN {X 0,Y 215.641,Z 373.449,A -85,B 0,C 180,E1 -23444.532,E2 -23444.532} C_VEL
LIN {X 0,Y 211.932,Z 386.633,A -85,B 0,C 180,E1 -23445.536,E2 -23445.536} C_VEL
LIN {X 0,Y 207.626,Z 398.398,A -85,B 0,C 180,E1 -23446.735,E2 -23446.735} C_VEL
LIN {X 0,Y 202.91,Z 409.162,A -85,B 0,C 180,E1 -23448.189,E2 -23448.189} C_VEL
LIN {X 0,Y 201.518,Z 412.109,A -85,B 0,C 180,E1 -23448.685,E2 -23448.685} C_VEL
LIN {X 0,Y 198.811,Z 416.798,A -85,B 0,C 180,E1 -23449.386,E2 -23449.386} C_VEL
LIN {X 0,Y 192.936,Z 424.205,A -85,B 0,C 180,E1 -23450.247,E2 -23450.247} C_VEL
LIN {X 0,Y 186.748,Z 431.112,A -85,B 0,C 180,E1 -23451.286,E2 -23451.286} C_VEL
LIN {X 0,Y 183.6,Z 434.911,A -85,B 0,C 180,E1 -23452.278,E2 -23452.278} C_VEL
LIN {X 0,Y 176.965,Z 443.547,A -85,B 0,C 180,E1 -23455.538,E2 -23455.538} C_VEL
LIN {X 0,Y 171.1,Z 450.497,A -85,B 0,C 180,E1 -23459.11,E2 -23459.11} C_VEL
LIN {X 0,Y 166.766,Z 455.164,A -85,B 0,C 180,E1 -23462.385,E2 -23462.385} C_VEL
LIN {X 0,Y 163.052,Z 458.796,A -85,B 0,C 180,E1 -23465.831,E2 -23465.831} C_VEL
LIN {X 0,Y 159.987,Z 461.499,A -85,B 0,C 180,E1 -23469.427,E2 -23469.427} C_VEL
LIN {X 0,Y 158.274,Z 462.836,A -85,B 0,C 180,E1 -23471.893,E2 -23471.893} C_VEL
LIN {X 0,Y 156.936,Z 463.769,A -85,B 0,C 180,E1 -23474.415,E2 -23474.415} C_VEL
LIN {X 0,Y 155.37,Z 464.484,A -85,B 0,C 180,E1 -23479.577,E2 -23479.577} C_VEL
LIN {X 0,Y 154.909,Z 463.719,A -85,B 0,C 180,E1 -23484.794,E2 -23484.794} C_VEL
LIN {X 0,Y 155.087,Z 462.734,A -85,B 0,C 180,E1 -23487.403,E2 -23487.403} C_VEL
LIN {X 0,Y 155.244,Z 461.298,A -85,B 0,C 180,E1 -23490,E2 -23490} C_VEL
LIN {X 0,Y 155.151,Z 458.739,A -85,B 0,C 180,E1 -23493.379,E2 -23493.379} C_VEL
LIN {X 0,Y 155.177,Z 455.584,A -85,B 0,C 180,E1 -23496.5,E2 -23496.5} C_VEL
LIN {X 0,Y 155.553,Z 450.565,A -85,B 0,C 180,E1 -23500.41,E2 -23500.41} C_VEL
LIN {X 0,Y 156.438,Z 444.18,A -85,B 0,C 180,E1 -23504.303,E2 -23504.303} C_VEL
LIN {X 0,Y 158.029,Z 436.14,A -85,B 0,C 180,E1 -23508.136,E2 -23508.136} C_VEL
LIN {X 0,Y 159.729,Z 427.896,A -85,B 0,C 180,E1 -23511.282,E2 -23511.282} C_VEL
LIN {X 0,Y 161.982,Z 417.902,A -85,B 0,C 180,E1 -23514.335,E2 -23514.335} C_VEL
LIN {X 0,Y 164.392,Z 406.641,A -85,B 0,C 180,E1 -23517.012,E2 -23517.012} C_VEL
LIN {X 0,Y 166.834,Z 394.021,A -85,B 0,C 180,E1 -23519.318,E2 -23519.318} C_VEL
LIN {X 0,Y 168.872,Z 381.52,A -85,B 0,C 180,E1 -23520.994,E2 -23520.994} C_VEL
LIN {X 0,Y 170.592,Z 367.935,A -85,B 0,C 180,E1 -23522.291,E2 -23522.291} C_VEL
LIN {X 0,Y 171.661,Z 354.438,A -85,B 0,C 180,E1 -23523.11,E2 -23523.11} C_VEL
LIN {X 0,Y 173.821,Z 315.278,A -85,B 0,C 180,E1 -23525.038,E2 -23525.038} C_VEL
LIN {X 0,Y 171.258,Z 289.659,A -85,B 0,C 180,E1 -23526.883,E2 -23526.883} C_VEL
LIN {X 0,Y 164.093,Z 268.816,A -85,B 0,C 180,E1 -23529.262,E2 -23529.262} C_VEL
LIN {X 0,Y 158.936,Z 255.753,A -85,B 0,C 180,E1 -23531.018,E2 -23531.018} C_VEL
LIN {X 0,Y 157.963,Z 253.064,A -85,B 0,C 180,E1 -23531.48,E2 -23531.48} C_VEL
LIN {X 0,Y 157.233,Z 249.904,A -85,B 0,C 180,E1 -23533.523,E2 -23533.523} C_VEL
LIN {X 0,Y 157.185,Z 249.908,A -85,B 0,C 180,E1 -23539.465,E2 -23539.465} C_VEL
LIN {X 0,Y 157.262,Z 249.893,A -85,B 0,C 180,E1 -23544.48,E2 -23544.48} C_VEL
LIN {X 0,Y 157.27,Z 249.896,A -85,B 0,C 180,E1 -23548.099,E2 -23548.099} C_VEL
LIN {X 0,Y 157.296,Z 249.88,A -85,B 0,C 180,E1 -23553.46,E2 -23553.46} C_VEL
LIN {X 0,Y 157.344,Z 249.884,A -85,B 0,C 180,E1 -23559.7,E2 -23559.7} C_VEL
LIN {X 0,Y 157.394,Z 249.857,A -85,B 0,C 180,E1 -23564.459,E2 -23564.459} C_VEL
LIN {X 0,Y 157.667,Z 249.845,A -85,B 0,C 180,E1 -23569.728,E2 -23569.728} C_VEL
LIN {X 0,Y 157.739,Z 249.835,A -85,B 0,C 180,E1 -23572.318,E2 -23572.318} C_VEL
LIN {X 0,Y 158.223,Z 249.744,A -85,B 0,C 180,E1 -23579.999,E2 -23579.999} C_VEL
LIN {X 0,Y 157.739,Z 249.835,A -85,B 0,C 180,E1 -23587.68,E2 -23587.68} C_VEL
LIN {X 0,Y 157.613,Z 249.846,A -85,B 0,C 180,E1 -23591.225,E2 -23591.225} C_VEL
LIN {X 0,Y 157.425,Z 249.849,A -85,B 0,C 180,E1 -23595.536,E2 -23595.536} C_VEL
LIN {X 0,Y 157.369,Z 249.848,A -85,B 0,C 180,E1 -23600.932,E2 -23600.932} C_VEL
LIN {X 0,Y 157.298,Z 249.888,A -85,B 0,C 180,E1 -23606.685,E2 -23606.685} C_VEL
LIN {X 0,Y 157.261,Z 249.89,A -85,B 0,C 180,E1 -23612.43,E2 -23612.43} C_VEL
LIN {X 0,Y 157.269,Z 249.87,A -85,B 0,C 180,E1 -23616.459,E2 -23616.459} C_VEL
LIN {X 0,Y 157.223,Z 249.873,A -85,B 0,C 180,E1 -23622.105,E2 -23622.105} C_VEL
LIN {X 0,Y 157.201,Z 249.902,A -85,B 0,C 180,E1 -23627.892,E2 -23627.892} C_VEL
LIN {X 0,Y 157.258,Z 249.887,A -85,B 0,C 180,E1 -23633.554,E2 -23633.554} C_VEL
LIN {X 0,Y 157.285,Z 249.865,A -85,B 0,C 180,E1 -23638.099,E2 -23638.099} C_VEL
LIN {X 0,Y 157.316,Z 249.888,A -85,B 0,C 180,E1 -23643.468,E2 -23643.468} C_VEL
LIN {X 0,Y 157.39,Z 249.866,A -85,B 0,C 180,E1 -23649.67,E2 -23649.67} C_VEL
LIN {X 0,Y 157.475,Z 249.866,A -85,B 0,C 180,E1 -23654.47,E2 -23654.47} C_VEL
LIN {X 0,Y 157.724,Z 249.828,A -85,B 0,C 180,E1 -23659.734,E2 -23659.734} C_VEL
LIN {X 0,Y 157.802,Z 249.826,A -85,B 0,C 180,E1 -23662.323,E2 -23662.323} C_VEL
LIN {X 0,Y 158.256,Z 249.773,A -85,B 0,C 180,E1 -23670,E2 -23670} C_VEL
LIN {X 0,Y 157.794,Z 249.833,A -85,B 0,C 180,E1 -23677.678,E2 -23677.678} C_VEL
LIN {X 0,Y 157.744,Z 249.838,A -85,B 0,C 180,E1 -23679.293,E2 -23679.293} C_VEL
LIN {X 0,Y 158.88,Z 252.875,A -85,B 0,C 180,E1 -23679.748,E2 -23679.748} C_VEL
LIN {X 0,Y 168.407,Z 274.152,A -85,B 0,C 180,E1 -23682.734,E2 -23682.734} C_VEL
LIN {X 0,Y 174.894,Z 290.251,A -85,B 0,C 180,E1 -23684.638,E2 -23684.638} C_VEL
LIN {X 0,Y 171.273,Z 347.814,A -85,B 0,C 180,E1 -23687.48,E2 -23687.48} C_VEL
LIN {X 0,Y 170.101,Z 360.587,A -85,B 0,C 180,E1 -23688.539,E2 -23688.539} C_VEL
LIN {X 0,Y 168.563,Z 372.732,A -85,B 0,C 180,E1 -23689.958,E2 -23689.958} C_VEL
LIN {X 0,Y 166.581,Z 384.826,A -85,B 0,C 180,E1 -23691.851,E2 -23691.851} C_VEL
LIN {X 0,Y 164.29,Z 396.777,A -85,B 0,C 180,E1 -23694.294,E2 -23694.294} C_VEL
LIN {X 0,Y 162.059,Z 407.444,A -85,B 0,C 180,E1 -23697.085,E2 -23697.085} C_VEL
LIN {X 0,Y 159.862,Z 417.487,A -85,B 0,C 180,E1 -23700.43,E2 -23700.43} C_VEL
LIN {X 0,Y 157.942,Z 425.989,A -85,B 0,C 180,E1 -23703.98,E2 -23703.98} C_VEL
LIN {X 0,Y 156.537,Z 432.859,A -85,B 0,C 180,E1 -23707.585,E2 -23707.585} C_VEL
LIN {X 0,Y 155.536,Z 438.745,A -85,B 0,C 180,E1 -23711.477,E2 -23711.477} C_VEL
LIN {X 0,Y 154.84,Z 443.168,A -85,B 0,C 180,E1 -23715.184,E2 -23715.184} C_VEL
LIN {X 0,Y 154.509,Z 446.464,A -85,B 0,C 180,E1 -23718.736,E2 -23718.736} C_VEL
LIN {X 0,Y 154.779,Z 449.684,A -85,B 0,C 180,E1 -23723.824,E2 -23723.824} C_VEL
LIN {X 0,Y 155.987,Z 451.396,A -85,B 0,C 180,E1 -23728.865,E2 -23728.865} C_VEL
LIN {X 0,Y 158.011,Z 451.631,A -85,B 0,C 180,E1 -23733.592,E2 -23733.592} C_VEL
LIN {X 0,Y 160.16,Z 450.899,A -85,B 0,C 180,E1 -23737.132,E2 -23737.132} C_VEL
LIN {X 0,Y 163.351,Z 449.04,A -85,B 0,C 180,E1 -23741.16,E2 -23741.16} C_VEL
LIN {X 0,Y 167.763,Z 445.617,A -85,B 0,C 180,E1 -23745.443,E2 -23745.443} C_VEL
LIN {X 0,Y 171.995,Z 441.781,A -85,B 0,C 180,E1 -23748.688,E2 -23748.688} C_VEL
LIN {X 0,Y 177.329,Z 436.111,A -85,B 0,C 180,E1 -23752.182,E2 -23752.182} C_VEL
LIN {X 0,Y 183.282,Z 428.915,A -85,B 0,C 180,E1 -23755.466,E2 -23755.466} C_VEL
LIN {X 0,Y 189.395,Z 420.431,A -85,B 0,C 180,E1 -23758.299,E2 -23758.299} C_VEL
LIN {X 0,Y 195.526,Z 410.579,A -85,B 0,C 180,E1 -23760.767,E2 -23760.767} C_VEL
LIN {X 0,Y 200.97,Z 400.153,A -85,B 0,C 180,E1 -23762.758,E2 -23762.758} C_VEL
LIN {X 0,Y 205.921,Z 388.894,A -85,B 0,C 180,E1 -23764.405,E2 -23764.405} C_VEL
LIN {X 0,Y 210.275,Z 376.714,A -85,B 0,C 180,E1 -23765.755,E2 -23765.755} C_VEL
LIN {X 0,Y 213.466,Z 364.849,A -85,B 0,C 180,E1 -23766.766,E2 -23766.766} C_VEL
LIN {X 0,Y 216.162,Z 351.241,A -85,B 0,C 180,E1 -23767.553,E2 -23767.553} C_VEL
LIN {X 0,Y 219.553,Z 323.771,A -85,B 0,C 180,E1 -23768.612,E2 -23768.612} C_VEL
LIN {X 0,Y 218.022,Z 320.238,A -85,B 0,C 180,E1 -23770.034,E2 -23770.034} C_VEL
LIN {X 0,Y 214.925,Z 314.399,A -85,B 0,C 180,E1 -23773.314,E2 -23773.314} C_VEL
LIN {X 0,Y 214.02,Z 312.748,A -85,B 0,C 180,E1 -23774.524,E2 -23774.524} C_VEL
LIN {X 0,Y 212.147,Z 309.589,A -85,B 0,C 180,E1 -23777.515,E2 -23777.515} C_VEL
LIN {X 0,Y 210.645,Z 307.435,A -85,B 0,C 180,E1 -23781.532,E2 -23781.532} C_VEL
LIN {X 0,Y 210.303,Z 307.811,A -85,B 0,C 180,E1 -23786.364,E2 -23786.364} C_VEL
LIN {X 0,Y 210.924,Z 309.635,A -85,B 0,C 180,E1 -23789.487,E2 -23789.487} C_VEL
LIN {X 0,Y 212.813,Z 314.61,A -85,B 0,C 180,E1 -23793.726,E2 -23793.726} C_VEL
LIN {X 0,Y 214.572,Z 319.309,A -85,B 0,C 180,E1 -23796.378,E2 -23796.378} C_VEL
LIN {X 0,Y 216.596,Z 324.856,A -85,B 0,C 180,E1 -23798.767,E2 -23798.767} C_VEL
LIN {X 0,Y 218.708,Z 331.396,A -85,B 0,C 180,E1 -23800.947,E2 -23800.947} C_VEL
LIN {X 0,Y 218.842,Z 332.358,A -85,B 0,C 180,E1 -23801.133,E2 -23801.133} C_VEL
LIN {X 0,Y 215.299,Z 359.89,A -85,B 0,C 180,E1 -23802.146,E2 -23802.146} C_VEL
LIN {X 0,Y 212.575,Z 372.62,A -85,B 0,C 180,E1 -23802.781,E2 -23802.781} C_VEL
LIN {X 0,Y 208.948,Z 385.151,A -85,B 0,C 180,E1 -23803.691,E2 -23803.691} C_VEL
LIN {X 0,Y 204.524,Z 397.008,A -85,B 0,C 180,E1 -23804.874,E2 -23804.874} C_VEL
LIN {X 0,Y 198.973,Z 409.198,A -85,B 0,C 180,E1 -23806.473,E2 -23806.473} C_VEL
LIN {X 0,Y 193.223,Z 419.954,A -85,B 0,C 180,E1 -23808.415,E2 -23808.415} C_VEL
LIN {X 0,Y 187.798,Z 428.78,A -85,B 0,C 180,E1 -23810.496,E2 -23810.496} C_VEL
LIN {X 0,Y 183.6,Z 434.911,A -85,B 0,C 180,E1 -23812.278,E2 -23812.278} C_VEL
LIN {X 0,Y 180.412,Z 438.6,A -85,B 0,C 180,E1 -23813.375,E2 -23813.375} C_VEL
LIN {X 0,Y 171.189,Z 446.287,A -85,B 0,C 180,E1 -23815.65,E2 -23815.65} C_VEL
LIN {X 0,Y 166.281,Z 450.071,A -85,B 0,C 180,E1 -23817.287,E2 -23817.287} C_VEL
LIN {X 0,Y 164.384,Z 451.735,A -85,B 0,C 180,E1 -23818.31,E2 -23818.31} C_VEL
LIN {X 0,Y 159.182,Z 456.794,A -85,B 0,C 180,E1 -23822.385,E2 -23822.385} C_VEL
LIN {X 0,Y 155.424,Z 459.933,A -85,B 0,C 180,E1 -23825.988,E2 -23825.988} C_VEL
LIN {X 0,Y 153.357,Z 461.541,A -85,B 0,C 180,E1 -23828.495,E2 -23828.495} C_VEL
LIN {X 0,Y 150.075,Z 463.55,A -85,B 0,C 180,E1 -23833.683,E2 -23833.683} C_VEL
LIN {X 0,Y 148.357,Z 464.104,A -85,B 0,C 180,E1 -23839.078,E2 -23839.078} C_VEL
LIN {X 0,Y 147.926,Z 463.82,A -85,B 0,C 180,E1 -23841.806,E2 -23841.806} C_VEL
LIN {X 0,Y 148.014,Z 462.049,A -85,B 0,C 180,E1 -23847.279,E2 -23847.279} C_VEL
LIN {X 0,Y 148.184,Z 460.548,A -85,B 0,C 180,E1 -23850,E2 -23850} C_VEL
LIN {X 0,Y 148.161,Z 458.568,A -85,B 0,C 180,E1 -23852.718,E2 -23852.718} C_VEL
LIN {X 0,Y 148.122,Z 454.583,A -85,B 0,C 180,E1 -23856.811,E2 -23856.811} C_VEL
LIN {X 0,Y 148.688,Z 448.336,A -85,B 0,C 180,E1 -23861.587,E2 -23861.587} C_VEL
LIN {X 0,Y 149.8,Z 441.458,A -85,B 0,C 180,E1 -23865.648,E2 -23865.648} C_VEL
LIN {X 0,Y 151.267,Z 434.421,A -85,B 0,C 180,E1 -23868.977,E2 -23868.977} C_VEL
LIN {X 0,Y 153.092,Z 425.9,A -85,B 0,C 180,E1 -23872.252,E2 -23872.252} C_VEL
LIN {X 0,Y 155.225,Z 416.625,A -85,B 0,C 180,E1 -23875.104,E2 -23875.104} C_VEL
LIN {X 0,Y 157.758,Z 405.114,A -85,B 0,C 180,E1 -23877.886,E2 -23877.886} C_VEL
LIN {X 0,Y 160.001,Z 393.975,A -85,B 0,C 180,E1 -23879.972,E2 -23879.972} C_VEL
LIN {X 0,Y 162.078,Z 381.609,A -85,B 0,C 180,E1 -23881.715,E2 -23881.715} C_VEL
LIN {X 0,Y 163.958,Z 367.432,A -85,B 0,C 180,E1 -23883.124,E2 -23883.124} C_VEL
LIN {X 0,Y 165.058,Z 353.257,A -85,B 0,C 180,E1 -23884.01,E2 -23884.01} C_VEL
LIN {X 0,Y 167.271,Z 316.139,A -85,B 0,C 180,E1 -23885.905,E2 -23885.905} C_VEL
LIN {X 0,Y 164.914,Z 291.811,A -85,B 0,C 180,E1 -23887.714,E2 -23887.714} C_VEL
LIN {X 0,Y 158.362,Z 272.434,A -85,B 0,C 180,E1 -23890.043,E2 -23890.043} C_VEL
LIN {X 0,Y 153.069,Z 258.873,A -85,B 0,C 180,E1 -23891.941,E2 -23891.941} C_VEL
LIN {X 0,Y 150.648,Z 252.853,A -85,B 0,C 180,E1 -23892.876,E2 -23892.876} C_VEL
LIN {X 0,Y 150.141,Z 250.789,A -85,B 0,C 180,E1 -23894.294,E2 -23894.294} C_VEL
LIN {X 0,Y 150.127,Z 250.786,A -85,B 0,C 180,E1 -23899.049,E2 -23899.049} C_VEL
LIN {X 0,Y 150.165,Z 250.779,A -85,B 0,C 180,E1 -23902.706,E2 -23902.706} C_VEL
LIN {X 0,Y 150.195,Z 250.772,A -85,B 0,C 180,E1 -23907.369,E2 -23907.369} C_VEL
LIN {X 0,Y 150.226,Z 250.763,A -85,B 0,C 180,E1 -23912.719,E2 -23912.719} C_VEL
LIN {X 0,Y 150.268,Z 250.767,A -85,B 0,C 180,E1 -23919.274,E2 -23919.274} C_VEL
LIN {X 0,Y 150.298,Z 250.741,A -85,B 0,C 180,E1 -23923.705,E2 -23923.705} C_VEL
LIN {X 0,Y 150.587,Z 250.726,A -85,B 0,C 180,E1 -23929.24,E2 -23929.24} C_VEL
LIN {X 0,Y 150.662,Z 250.716,A -85,B 0,C 180,E1 -23931.955,E2 -23931.955} C_VEL
LIN {X 0,Y 151.183,Z 250.619,A -85,B 0,C 180,E1 -23939.999,E2 -23939.999} C_VEL
LIN {X 0,Y 150.662,Z 250.716,A -85,B 0,C 180,E1 -23948.044,E2 -23948.044} C_VEL
LIN {X 0,Y 150.555,Z 250.725,A -85,B 0,C 180,E1 -23951.427,E2 -23951.427} C_VEL
LIN {X 0,Y 150.34,Z 250.723,A -85,B 0,C 180,E1 -23956.288,E2 -23956.288} C_VEL
LIN {X 0,Y 150.351,Z 250.719,A -85,B 0,C 180,E1 -23960.809,E2 -23960.809} C_VEL
LIN {X 0,Y 150.228,Z 250.769,A -85,B 0,C 180,E1 -23967.283,E2 -23967.283} C_VEL
LIN {X 0,Y 150.202,Z 250.769,A -85,B 0,C 180,E1 -23972.634,E2 -23972.634} C_VEL
LIN {X 0,Y 150.2,Z 250.742,A -85,B 0,C 180,E1 -23977.464,E2 -23977.464} C_VEL
LIN {X 0,Y 150.162,Z 250.747,A -85,B 0,C 180,E1 -23981.517,E2 -23981.517} C_VEL
LIN {X 0,Y 150.126,Z 250.776,A -85,B 0,C 180,E1 -23985.402,E2 -23985.402} C_VEL
LIN {X 0,Y 150.141,Z 250.782,A -85,B 0,C 180,E1 -23989.061,E2 -23989.061} C_VEL
LIN {X 0,Y 150.17,Z 250.772,A -85,B 0,C 180,E1 -23992.711,E2 -23992.711} C_VEL
LIN {X 0,Y 150.207,Z 250.744,A -85,B 0,C 180,E1 -23997.371,E2 -23997.371} C_VEL
LIN {X 0,Y 150.238,Z 250.768,A -85,B 0,C 180,E1 -24002.721,E2 -24002.721} C_VEL
LIN {X 0,Y 150.347,Z 250.746,A -85,B 0,C 180,E1 -24009.21,E2 -24009.21} C_VEL
LIN {X 0,Y 150.379,Z 250.746,A -85,B 0,C 180,E1 -24013.717,E2 -24013.717} C_VEL
LIN {X 0,Y 150.65,Z 250.711,A -85,B 0,C 180,E1 -24019.247,E2 -24019.247} C_VEL
LIN {X 0,Y 150.737,Z 250.703,A -85,B 0,C 180,E1 -24021.961,E2 -24021.961} C_VEL
LIN {X 0,Y 151.217,Z 250.65,A -85,B 0,C 180,E1 -24030,E2 -24030} C_VEL
LIN {X 0,Y 150.74,Z 250.712,A -85,B 0,C 180,E1 -24037.955,E2 -24037.955} C_VEL
LIN {X 0,Y 151.839,Z 253.77,A -85,B 0,C 180,E1 -24038.442,E2 -24038.442} C_VEL
LIN {X 0,Y 161.456,Z 274.797,A -85,B 0,C 180,E1 -24041.613,E2 -24041.613} C_VEL
LIN {X 0,Y 168.343,Z 292.065,A -85,B 0,C 180,E1 -24043.787,E2 -24043.787} C_VEL
LIN {X 0,Y 164.593,Z 348.605,A -85,B 0,C 180,E1 -24046.687,E2 -24046.687} C_VEL
LIN {X 0,Y 163.406,Z 360.865,A -85,B 0,C 180,E1 -24047.744,E2 -24047.744} C_VEL
LIN {X 0,Y 161.665,Z 373.877,A -85,B 0,C 180,E1 -24049.331,E2 -24049.331} C_VEL
LIN {X 0,Y 159.395,Z 386.815,A -85,B 0,C 180,E1 -24051.496,E2 -24051.496} C_VEL
LIN {X 0,Y 157.411,Z 396.966,A -85,B 0,C 180,E1 -24053.69,E2 -24053.69} C_VEL
LIN {X 0,Y 155.103,Z 407.694,A -85,B 0,C 180,E1 -24056.604,E2 -24056.604} C_VEL
LIN {X 0,Y 152.967,Z 417.033,A -85,B 0,C 180,E1 -24059.813,E2 -24059.813} C_VEL
LIN {X 0,Y 151.113,Z 424.913,A -85,B 0,C 180,E1 -24063.162,E2 -24063.162} C_VEL
LIN {X 0,Y 149.604,Z 432.19,A -85,B 0,C 180,E1 -24067.004,E2 -24067.004} C_VEL
LIN {X 0,Y 148.413,Z 438.872,A -85,B 0,C 180,E1 -24071.521,E2 -24071.521} C_VEL
LIN {X 0,Y 147.705,Z 443.449,A -85,B 0,C 180,E1 -24075.532,E2 -24075.532} C_VEL
LIN {X 0,Y 147.397,Z 447.079,A -85,B 0,C 180,E1 -24079.713,E2 -24079.713} C_VEL
LIN {X 0,Y 147.715,Z 449.72,A -85,B 0,C 180,E1 -24083.973,E2 -24083.973} C_VEL
LIN {X 0,Y 148.776,Z 451.478,A -85,B 0,C 180,E1 -24088.694,E2 -24088.694} C_VEL
LIN {X 0,Y 150.322,Z 452.064,A -85,B 0,C 180,E1 -24092.649,E2 -24092.649} C_VEL
LIN {X 0,Y 152.753,Z 451.705,A -85,B 0,C 180,E1 -24096.938,E2 -24096.938} C_VEL
LIN {X 0,Y 156.425,Z 449.995,A -85,B 0,C 180,E1 -24101.67,E2 -24101.67} C_VEL
LIN {X 0,Y 159.909,Z 447.722,A -85,B 0,C 180,E1 -24105.193,E2 -24105.193} C_VEL
LIN {X 0,Y 164.656,Z 443.99,A -85,B 0,C 180,E1 -24108.993,E2 -24108.993} C_VEL
LIN {X 0,Y 170.603,Z 438.473,A -85,B 0,C 180,E1 -24112.902,E2 -24112.902} C_VEL
LIN {X 0,Y 176.625,Z 431.947,A -85,B 0,C 180,E1 -24116.218,E2 -24116.218} C_VEL
LIN {X 0,Y 182.733,Z 424.326,A -85,B 0,C 180,E1 -24119.051,E2 -24119.051} C_VEL
LIN {X 0,Y 189.069,Z 415.252,A -85,B 0,C 180,E1 -24121.599,E2 -24121.599} C_VEL
LIN {X 0,Y 194.721,Z 405.857,A -85,B 0,C 180,E1 -24123.622,E2 -24123.622} C_VEL
LIN {X 0,Y 200.02,Z 395.324,A -85,B 0,C 180,E1 -24125.374,E2 -24125.374} C_VEL
LIN {X 0,Y 204.963,Z 383.474,A -85,B 0,C 180,E1 -24126.867,E2 -24126.867} C_VEL
LIN {X 0,Y 208.807,Z 371.643,A -85,B 0,C 180,E1 -24128.02,E2 -24128.02} C_VEL
LIN {X 0,Y 212.094,Z 358.174,A -85,B 0,C 180,E1 -24128.947,E2 -24128.947} C_VEL
LIN {X 0,Y 214.294,Z 345.014,A -85,B 0,C 180,E1 -24129.538,E2 -24129.538} C_VEL
LIN {X 0,Y 216.496,Z 327.641,A -85,B 0,C 180,E1 -24130.18,E2 -24130.18} C_VEL
LIN {X 0,Y 213.301,Z 321.149,A -85,B 0,C 180,E1 -24133.759,E2 -24133.759} C_VEL
LIN {X 0,Y 212.279,Z 319.279,A -85,B 0,C 180,E1 -24135.196,E2 -24135.196} C_VEL
LIN {X 0,Y 210.797,Z 316.487,A -85,B 0,C 180,E1 -24137.799,E2 -24137.799} C_VEL
LIN {X 0,Y 209.43,Z 314.435,A -85,B 0,C 180,E1 -24141.663,E2 -24141.663} C_VEL
LIN {X 0,Y 209.11,Z 314.819,A -85,B 0,C 180,E1 -24146.301,E2 -24146.301} C_VEL
LIN {X 0,Y 209.631,Z 316.568,A -85,B 0,C 180,E1 -24149.231,E2 -24149.231} C_VEL
LIN {X 0,Y 211.285,Z 321.464,A -85,B 0,C 180,E1 -24153.315,E2 -24153.315} C_VEL
LIN {X 0,Y 212.663,Z 325.494,A -85,B 0,C 180,E1 -24155.601,E2 -24155.601} C_VEL
LIN {X 0,Y 214.592,Z 331.297,A -85,B 0,C 180,E1 -24158.114,E2 -24158.114} C_VEL
LIN {X 0,Y 215.697,Z 335.263,A -85,B 0,C 180,E1 -24159.462,E2 -24159.462} C_VEL
LIN {X 0,Y 212.319,Z 360.368,A -85,B 0,C 180,E1 -24160.426,E2 -24160.426} C_VEL
LIN {X 0,Y 209.504,Z 372.891,A -85,B 0,C 180,E1 -24161.044,E2 -24161.044} C_VEL
LIN {X 0,Y 205.588,Z 385.722,A -85,B 0,C 180,E1 -24161.975,E2 -24161.975} C_VEL
LIN {X 0,Y 200.367,Z 398.904,A -85,B 0,C 180,E1 -24163.303,E2 -24163.303} C_VEL
LIN {X 0,Y 194.636,Z 410.535,A -85,B 0,C 180,E1 -24164.883,E2 -24164.883} C_VEL
LIN {X 0,Y 189.233,Z 419.96,A -85,B 0,C 180,E1 -24166.606,E2 -24166.606} C_VEL
LIN {X 0,Y 182.48,Z 430.293,A -85,B 0,C 180,E1 -24169.106,E2 -24169.106} C_VEL
LIN {X 0,Y 176.147,Z 438.668,A -85,B 0,C 180,E1 -24171.803,E2 -24171.803} C_VEL
LIN {X 0,Y 170.288,Z 445.501,A -85,B 0,C 180,E1 -24174.709,E2 -24174.709} C_VEL
LIN {X 0,Y 164.384,Z 451.735,A -85,B 0,C 180,E1 -24178.31,E2 -24178.31} C_VEL
LIN {X 0,Y 161.424,Z 454.146,A -85,B 0,C 180,E1 -24179.908,E2 -24179.908} C_VEL
LIN {X 0,Y 155.222,Z 457.553,A -85,B 0,C 180,E1 -24182.433,E2 -24182.433} C_VEL
LIN {X 0,Y 149.32,Z 460.206,A -85,B 0,C 180,E1 -24185.25,E2 -24185.25} C_VEL
LIN {X 0,Y 146.906,Z 461.398,A -85,B 0,C 180,E1 -24187.266,E2 -24187.266} C_VEL
LIN {X 0,Y 144.815,Z 462.611,A -85,B 0,C 180,E1 -24190.142,E2 -24190.142} C_VEL
LIN {X 0,Y 142.148,Z 463.714,A -85,B 0,C 180,E1 -24195.689,E2 -24195.689} C_VEL
LIN {X 0,Y 140.909,Z 463.286,A -85,B 0,C 180,E1 -24201.395,E2 -24201.395} C_VEL
LIN {X 0,Y 140.915,Z 461.343,A -85,B 0,C 180,E1 -24207.141,E2 -24207.141} C_VEL
LIN {X 0,Y 141.125,Z 459.756,A -85,B 0,C 180,E1 -24210,E2 -24210} C_VEL
LIN {X 0,Y 141.107,Z 457.626,A -85,B 0,C 180,E1 -24212.854,E2 -24212.854} C_VEL
LIN {X 0,Y 141.074,Z 453.468,A -85,B 0,C 180,E1 -24217.153,E2 -24217.153} C_VEL
LIN {X 0,Y 141.735,Z 447.042,A -85,B 0,C 180,E1 -24222.164,E2 -24222.164} C_VEL
LIN {X 0,Y 142.965,Z 439.947,A -85,B 0,C 180,E1 -24226.417,E2 -24226.417} C_VEL
LIN {X 0,Y 144.547,Z 432.658,A -85,B 0,C 180,E1 -24229.895,E2 -24229.895} C_VEL
LIN {X 0,Y 146.569,Z 423.795,A -85,B 0,C 180,E1 -24233.3,E2 -24233.3} C_VEL
LIN {X 0,Y 148.84,Z 413.944,A -85,B 0,C 180,E1 -24236.32,E2 -24236.32} C_VEL
LIN {X 0,Y 151.162,Z 403.587,A -85,B 0,C 180,E1 -24238.836,E2 -24238.836} C_VEL
LIN {X 0,Y 153.525,Z 392.085,A -85,B 0,C 180,E1 -24240.993,E2 -24240.993} C_VEL
LIN {X 0,Y 155.699,Z 379.232,A -85,B 0,C 180,E1 -24242.792,E2 -24242.792} C_VEL
LIN {X 0,Y 157.442,Z 365.83,A -85,B 0,C 180,E1 -24244.105,E2 -24244.105} C_VEL
LIN {X 0,Y 158.69,Z 348.778,A -85,B 0,C 180,E1 -24245.147,E2 -24245.147} C_VEL
LIN {X 0,Y 160.691,Z 316.679,A -85,B 0,C 180,E1 -24246.846,E2 -24246.846} C_VEL
LIN {X 0,Y 158.526,Z 293.709,A -85,B 0,C 180,E1 -24248.645,E2 -24248.645} C_VEL
LIN {X 0,Y 152.304,Z 275.093,A -85,B 0,C 180,E1 -24250.995,E2 -24250.995} C_VEL
LIN {X 0,Y 146.457,Z 260.055,A -85,B 0,C 180,E1 -24253.213,E2 -24253.213} C_VEL
LIN {X 0,Y 143.239,Z 252.478,A -85,B 0,C 180,E1 -24254.514,E2 -24254.514} C_VEL
LIN {X 0,Y 143.078,Z 251.669,A -85,B 0,C 180,E1 -24255.08,E2 -24255.08} C_VEL
LIN {X 0,Y 143.061,Z 251.664,A -85,B 0,C 180,E1 -24261.806,E2 -24261.806} C_VEL
LIN {X 0,Y 143.163,Z 251.648,A -85,B 0,C 180,E1 -24267.315,E2 -24267.315} C_VEL
LIN {X 0,Y 143.17,Z 251.645,A -85,B 0,C 180,E1 -24272.066,E2 -24272.066} C_VEL
LIN {X 0,Y 143.207,Z 251.647,A -85,B 0,C 180,E1 -24278.801,E2 -24278.801} C_VEL
LIN {X 0,Y 143.238,Z 251.623,A -85,B 0,C 180,E1 -24282.878,E2 -24282.878} C_VEL
LIN {X 0,Y 143.514,Z 251.605,A -85,B 0,C 180,E1 -24288.703,E2 -24288.703} C_VEL
LIN {X 0,Y 143.588,Z 251.598,A -85,B 0,C 180,E1 -24291.555,E2 -24291.555} C_VEL
LIN {X 0,Y 144.141,Z 251.495,A -85,B 0,C 180,E1 -24299.999,E2 -24299.999} C_VEL
LIN {X 0,Y 143.588,Z 251.599,A -85,B 0,C 180,E1 -24308.443,E2 -24308.443} C_VEL
LIN {X 0,Y 143.482,Z 251.605,A -85,B 0,C 180,E1 -24311.616,E2 -24311.616} C_VEL
LIN {X 0,Y 143.286,Z 251.594,A -85,B 0,C 180,E1 -24317.114,E2 -24317.114} C_VEL
LIN {X 0,Y 143.278,Z 251.602,A -85,B 0,C 180,E1 -24321.271,E2 -24321.271} C_VEL
LIN {X 0,Y 143.175,Z 251.648,A -85,B 0,C 180,E1 -24327.937,E2 -24327.937} C_VEL
LIN {X 0,Y 143.153,Z 251.645,A -85,B 0,C 180,E1 -24333.435,E2 -24333.435} C_VEL
LIN {X 0,Y 143.074,Z 251.618,A -85,B 0,C 180,E1 -24339.685,E2 -24339.685} C_VEL
LIN {X 0,Y 143.061,Z 251.646,A -85,B 0,C 180,E1 -24343.452,E2 -24343.452} C_VEL
LIN {X 0,Y 143.058,Z 251.662,A -85,B 0,C 180,E1 -24347.467,E2 -24347.467} C_VEL
LIN {X 0,Y 143.069,Z 251.66,A -85,B 0,C 180,E1 -24351.809,E2 -24351.809} C_VEL
LIN {X 0,Y 143.174,Z 251.619,A -85,B 0,C 180,E1 -24357.324,E2 -24357.324} C_VEL
LIN {X 0,Y 143.184,Z 251.643,A -85,B 0,C 180,E1 -24362.066,E2 -24362.066} C_VEL
LIN {X 0,Y 143.273,Z 251.63,A -85,B 0,C 180,E1 -24368.748,E2 -24368.748} C_VEL
LIN {X 0,Y 143.313,Z 251.622,A -85,B 0,C 180,E1 -24372.89,E2 -24372.89} C_VEL
LIN {X 0,Y 143.592,Z 251.594,A -85,B 0,C 180,E1 -24378.711,E2 -24378.711} C_VEL
LIN {X 0,Y 143.658,Z 251.582,A -85,B 0,C 180,E1 -24381.562,E2 -24381.562} C_VEL
LIN {X 0,Y 144.175,Z 251.527,A -85,B 0,C 180,E1 -24390,E2 -24390} C_VEL
LIN {X 0,Y 143.632,Z 251.591,A -85,B 0,C 180,E1 -24396.497,E2 -24396.497} C_VEL
LIN {X 0,Y 144.708,Z 254.468,A -85,B 0,C 180,E1 -24396.973,E2 -24396.973} C_VEL
LIN {X 0,Y 150.304,Z 266.163,A -85,B 0,C 180,E1 -24398.989,E2 -24398.989} C_VEL
LIN {X 0,Y 157.279,Z 282.305,A -85,B 0,C 180,E1 -24401.354,E2 -24401.354} C_VEL
LIN {X 0,Y 161.816,Z 294.041,A -85,B 0,C 180,E1 -24402.88,E2 -24402.88} C_VEL
LIN {X 0,Y 158,Z 348.629,A -85,B 0,C 180,E1 -24405.767,E2 -24405.767} C_VEL
LIN {X 0,Y 156.708,Z 361.38,A -85,B 0,C 180,E1 -24406.905,E2 -24406.905} C_VEL
LIN {X 0,Y 154.935,Z 374.077,A -85,B 0,C 180,E1 -24408.512,E2 -24408.512} C_VEL
LIN {X 0,Y 152.618,Z 386.893,A -85,B 0,C 180,E1 -24410.73,E2 -24410.73} C_VEL
LIN {X 0,Y 150.222,Z 398.739,A -85,B 0,C 180,E1 -24413.428,E2 -24413.428} C_VEL
LIN {X 0,Y 147.927,Z 408.816,A -85,B 0,C 180,E1 -24416.379,E2 -24416.379} C_VEL
LIN {X 0,Y 145.729,Z 418.065,A -85,B 0,C 180,E1 -24419.766,E2 -24419.766} C_VEL
LIN {X 0,Y 143.645,Z 426.699,A -85,B 0,C 180,E1 -24423.724,E2 -24423.724} C_VEL
LIN {X 0,Y 142.207,Z 433.634,A -85,B 0,C 180,E1 -24427.748,E2 -24427.748} C_VEL
LIN {X 0,Y 141.233,Z 439.119,A -85,B 0,C 180,E1 -24431.72,E2 -24431.72} C_VEL
LIN {X 0,Y 140.592,Z 443.392,A -85,B 0,C 180,E1 -24435.587,E2 -24435.587} C_VEL
LIN {X 0,Y 140.312,Z 446.658,A -85,B 0,C 180,E1 -24439.373,E2 -24439.373} C_VEL
LIN {X 0,Y 140.511,Z 449.156,A -85,B 0,C 180,E1 -24443.149,E2 -24443.149} C_VEL
LIN {X 0,Y 141.345,Z 451.211,A -85,B 0,C 180,E1 -24447.692,E2 -24447.692} C_VEL
LIN {X 0,Y 142.946,Z 452.274,A -85,B 0,C 180,E1 -24452.237,E2 -24452.237} C_VEL
LIN {X 0,Y 145.701,Z 452.255,A -85,B 0,C 180,E1 -24457.302,E2 -24457.302} C_VEL
LIN {X 0,Y 148.543,Z 451.333,A -85,B 0,C 180,E1 -24461.112,E2 -24461.112} C_VEL
LIN {X 0,Y 152.523,Z 449.245,A -85,B 0,C 180,E1 -24465.362,E2 -24465.362} C_VEL
LIN {X 0,Y 157.902,Z 445.625,A -85,B 0,C 180,E1 -24469.746,E2 -24469.746} C_VEL
LIN {X 0,Y 164.62,Z 440.036,A -85,B 0,C 180,E1 -24474.097,E2 -24474.097} C_VEL
LIN {X 0,Y 171.22,Z 433.45,A -85,B 0,C 180,E1 -24477.648,E2 -24477.648} C_VEL
LIN {X 0,Y 177.767,Z 426.022,A -85,B 0,C 180,E1 -24480.567,E2 -24480.567} C_VEL
LIN {X 0,Y 184.432,Z 417.146,A -85,B 0,C 180,E1 -24483.147,E2 -24483.147} C_VEL
LIN {X 0,Y 190.535,Z 407.626,A -85,B 0,C 180,E1 -24485.251,E2 -24485.251} C_VEL
LIN {X 0,Y 195.854,Z 397.835,A -85,B 0,C 180,E1 -24486.926,E2 -24486.926} C_VEL
LIN {X 0,Y 201.397,Z 385.501,A -85,B 0,C 180,E1 -24488.53,E2 -24488.53} C_VEL
LIN {X 0,Y 205.694,Z 373.442,A -85,B 0,C 180,E1 -24489.713,E2 -24489.713} C_VEL
LIN {X 0,Y 209.06,Z 360.79,A -85,B 0,C 180,E1 -24490.624,E2 -24490.624} C_VEL
LIN {X 0,Y 211.376,Z 348.486,A -85,B 0,C 180,E1 -24491.209,E2 -24491.209} C_VEL
LIN {X 0,Y 213.532,Z 332.066,A -85,B 0,C 180,E1 -24491.846,E2 -24491.846} C_VEL
LIN {X 0,Y 211.226,Z 326.787,A -85,B 0,C 180,E1 -24494.915,E2 -24494.915} C_VEL
LIN {X 0,Y 209.315,Z 323.125,A -85,B 0,C 180,E1 -24498.4,E2 -24498.4} C_VEL
LIN {X 0,Y 208.214,Z 321.435,A -85,B 0,C 180,E1 -24501.796,E2 -24501.796} C_VEL
LIN {X 0,Y 207.902,Z 321.772,A -85,B 0,C 180,E1 -24506.07,E2 -24506.07} C_VEL
LIN {X 0,Y 208.258,Z 323.264,A -85,B 0,C 180,E1 -24508.68,E2 -24508.68} C_VEL
LIN {X 0,Y 209.68,Z 328.04,A -85,B 0,C 180,E1 -24512.728,E2 -24512.728} C_VEL
LIN {X 0,Y 210.968,Z 332.237,A -85,B 0,C 180,E1 -24515.061,E2 -24515.061} C_VEL
LIN {X 0,Y 212.541,Z 337.521,A -85,B 0,C 180,E1 -24517.358,E2 -24517.358} C_VEL
LIN {X 0,Y 212.885,Z 338.986,A -85,B 0,C 180,E1 -24517.842,E2 -24517.842} C_VEL
LIN {X 0,Y 209.796,Z 360.218,A -85,B 0,C 180,E1 -24518.614,E2 -24518.614} C_VEL
LIN {X 0,Y 206.552,Z 373.852,A -85,B 0,C 180,E1 -24519.286,E2 -24519.286} C_VEL
LIN {X 0,Y 202.422,Z 386.413,A -85,B 0,C 180,E1 -24520.204,E2 -24520.204} C_VEL
LIN {X 0,Y 197.033,Z 399.301,A -85,B 0,C 180,E1 -24521.499,E2 -24521.499} C_VEL
LIN {X 0,Y 191.107,Z 410.762,A -85,B 0,C 180,E1 -24523.044,E2 -24523.044} C_VEL
LIN {X 0,Y 184.274,Z 421.998,A -85,B 0,C 180,E1 -24525.131,E2 -24525.131} C_VEL
LIN {X 0,Y 177.272,Z 431.776,A -85,B 0,C 180,E1 -24527.631,E2 -24527.631} C_VEL
LIN {X 0,Y 170.696,Z 439.756,A -85,B 0,C 180,E1 -24530.349,E2 -24530.349} C_VEL
LIN {X 0,Y 164.601,Z 446.337,A -85,B 0,C 180,E1 -24533.295,E2 -24533.295} C_VEL
LIN {X 0,Y 158.296,Z 452.4,A -85,B 0,C 180,E1 -24537.041,E2 -24537.041} C_VEL
LIN {X 0,Y 153.458,Z 456.641,A -85,B 0,C 180,E1 -24540.678,E2 -24540.678} C_VEL
LIN {X 0,Y 148.954,Z 460.044,A -85,B 0,C 180,E1 -24544.875,E2 -24544.875} C_VEL
LIN {X 0,Y 146.906,Z 461.398,A -85,B 0,C 180,E1 -24547.266,E2 -24547.266} C_VEL
LIN {X 0,Y 144.676,Z 462.411,A -85,B 0,C 180,E1 -24549.379,E2 -24549.379} C_VEL
LIN {X 0,Y 139.767,Z 463.302,A -85,B 0,C 180,E1 -24552.832,E2 -24552.832} C_VEL
LIN {X 0,Y 136.137,Z 463.408,A -85,B 0,C 180,E1 -24555.768,E2 -24555.768} C_VEL
LIN {X 0,Y 134.43,Z 463.202,A -85,B 0,C 180,E1 -24558.165,E2 -24558.165} C_VEL
LIN {X 0,Y 134.175,Z 463.048,A -85,B 0,C 180,E1 -24558.997,E2 -24558.997} C_VEL
LIN {X 0,Y 133.739,Z 461.881,A -85,B 0,C 180,E1 -24563.967,E2 -24563.967} C_VEL
LIN {X 0,Y 133.848,Z 460.622,A -85,B 0,C 180,E1 -24566.99,E2 -24566.99} C_VEL
LIN {X 0,Y 134.067,Z 458.891,A -85,B 0,C 180,E1 -24570,E2 -24570} C_VEL
LIN {X 0,Y 134.054,Z 456.663,A -85,B 0,C 180,E1 -24573.005,E2 -24573.005} C_VEL
LIN {X 0,Y 134.055,Z 452.315,A -85,B 0,C 180,E1 -24577.53,E2 -24577.53} C_VEL
LIN {X 0,Y 134.628,Z 446.698,A -85,B 0,C 180,E1 -24582.051,E2 -24582.051} C_VEL
LIN {X 0,Y 135.881,Z 439.606,A -85,B 0,C 180,E1 -24586.525,E2 -24586.525} C_VEL
LIN {X 0,Y 137.844,Z 430.681,A -85,B 0,C 180,E1 -24590.907,E2 -24590.907} C_VEL
LIN {X 0,Y 140.06,Z 421.542,A -85,B 0,C 180,E1 -24594.451,E2 -24594.451} C_VEL
LIN {X 0,Y 142.345,Z 411.873,A -85,B 0,C 180,E1 -24597.434,E2 -24597.434} C_VEL
LIN {X 0,Y 144.628,Z 401.899,A -85,B 0,C 180,E1 -24599.869,E2 -24599.869} C_VEL
LIN {X 0,Y 147.125,Z 390.079,A -85,B 0,C 180,E1 -24602.098,E2 -24602.098} C_VEL
LIN {X 0,Y 149.18,Z 378.029,A -85,B 0,C 180,E1 -24603.809,E2 -24603.809} C_VEL
LIN {X 0,Y 150.984,Z 364.172,A -85,B 0,C 180,E1 -24605.167,E2 -24605.167} C_VEL
LIN {X 0,Y 152.466,Z 343.867,A -85,B 0,C 180,E1 -24606.399,E2 -24606.399} C_VEL
LIN {X 0,Y 154.174,Z 317.299,A -85,B 0,C 180,E1 -24607.86,E2 -24607.86} C_VEL
LIN {X 0,Y 152.257,Z 295.947,A -85,B 0,C 180,E1 -24609.6,E2 -24609.6} C_VEL
LIN {X 0,Y 146.368,Z 278.159,A -85,B 0,C 180,E1 -24611.936,E2 -24611.936} C_VEL
LIN {X 0,Y 141.26,Z 264.749,A -85,B 0,C 180,E1 -24614.015,E2 -24614.015} C_VEL
LIN {X 0,Y 137.31,Z 255.821,A -85,B 0,C 180,E1 -24615.628,E2 -24615.628} C_VEL
LIN {X 0,Y 136.057,Z 252.941,A -85,B 0,C 180,E1 -24616.158,E2 -24616.158} C_VEL
LIN {X 0,Y 136.006,Z 252.549,A -85,B 0,C 180,E1 -24616.332,E2 -24616.332} C_VEL
LIN {X 0,Y 136.01,Z 252.542,A -85,B 0,C 180,E1 -24621.677,E2 -24621.677} C_VEL
LIN {X 0,Y 136.041,Z 252.531,A -85,B 0,C 180,E1 -24625.738,E2 -24625.738} C_VEL
LIN {X 0,Y 136.111,Z 252.522,A -85,B 0,C 180,E1 -24632.307,E2 -24632.307} C_VEL
LIN {X 0,Y 136.17,Z 252.523,A -85,B 0,C 180,E1 -24638.82,E2 -24638.82} C_VEL
LIN {X 0,Y 136.208,Z 252.495,A -85,B 0,C 180,E1 -24645.048,E2 -24645.048} C_VEL
LIN {X 0,Y 136.411,Z 252.489,A -85,B 0,C 180,E1 -24648.177,E2 -24648.177} C_VEL
LIN {X 0,Y 136.517,Z 252.481,A -85,B 0,C 180,E1 -24651.114,E2 -24651.114} C_VEL
LIN {X 0,Y 137.098,Z 252.371,A -85,B 0,C 180,E1 -24659.999,E2 -24659.999} C_VEL
LIN {X 0,Y 136.517,Z 252.479,A -85,B 0,C 180,E1 -24668.883,E2 -24668.883} C_VEL
LIN {X 0,Y 136.399,Z 252.487,A -85,B 0,C 180,E1 -24671.893,E2 -24671.893} C_VEL
LIN {X 0,Y 136.205,Z 252.468,A -85,B 0,C 180,E1 -24678.033,E2 -24678.033} C_VEL
LIN {X 0,Y 136.197,Z 252.487,A -85,B 0,C 180,E1 -24681.764,E2 -24681.764} C_VEL
LIN {X 0,Y 136.085,Z 252.534,A -85,B 0,C 180,E1 -24688.616,E2 -24688.616} C_VEL
LIN {X 0,Y 136.065,Z 252.52,A -85,B 0,C 180,E1 -24694.621,E2 -24694.621} C_VEL
LIN {X 0,Y 136.046,Z 252.491,A -85,B 0,C 180,E1 -24699.214,E2 -24699.214} C_VEL
LIN {X 0,Y 136,Z 252.525,A -85,B 0,C 180,E1 -24703.665,E2 -24703.665} C_VEL
LIN {X 0,Y 135.997,Z 252.543,A -85,B 0,C 180,E1 -24707.799,E2 -24707.799} C_VEL
LIN {X 0,Y 136.018,Z 252.539,A -85,B 0,C 180,E1 -24711.687,E2 -24711.687} C_VEL
LIN {X 0,Y 136.047,Z 252.512,A -85,B 0,C 180,E1 -24715.743,E2 -24715.743} C_VEL
LIN {X 0,Y 136.141,Z 252.522,A -85,B 0,C 180,E1 -24722.319,E2 -24722.319} C_VEL
LIN {X 0,Y 136.24,Z 252.505,A -85,B 0,C 180,E1 -24728.835,E2 -24728.835} C_VEL
LIN {X 0,Y 136.281,Z 252.507,A -85,B 0,C 180,E1 -24735.059,E2 -24735.059} C_VEL
LIN {X 0,Y 136.495,Z 252.479,A -85,B 0,C 180,E1 -24738.116,E2 -24738.116} C_VEL
LIN {X 0,Y 136.586,Z 252.46,A -85,B 0,C 180,E1 -24741.121,E2 -24741.121} C_VEL
LIN {X 0,Y 137.132,Z 252.404,A -85,B 0,C 180,E1 -24750,E2 -24750} C_VEL
LIN {X 0,Y 136.601,Z 252.471,A -85,B 0,C 180,E1 -24754.888,E2 -24754.888} C_VEL
LIN {X 0,Y 137.623,Z 255.391,A -85,B 0,C 180,E1 -24755.402,E2 -24755.402} C_VEL
LIN {X 0,Y 142.531,Z 264.987,A -85,B 0,C 180,E1 -24757.257,E2 -24757.257} C_VEL
LIN {X 0,Y 150.72,Z 283.882,A -85,B 0,C 180,E1 -24760.282,E2 -24760.282} C_VEL
LIN {X 0,Y 155.207,Z 295.315,A -85,B 0,C 180,E1 -24761.844,E2 -24761.844} C_VEL
LIN {X 0,Y 151.401,Z 348.522,A -85,B 0,C 180,E1 -24764.782,E2 -24764.782} C_VEL
LIN {X 0,Y 149.966,Z 362.273,A -85,B 0,C 180,E1 -24766.067,E2 -24766.067} C_VEL
LIN {X 0,Y 148.161,Z 374.61,A -85,B 0,C 180,E1 -24767.713,E2 -24767.713} C_VEL
LIN {X 0,Y 145.643,Z 387.759,A -85,B 0,C 180,E1 -24770.106,E2 -24770.106} C_VEL
LIN {X 0,Y 143.285,Z 399.02,A -85,B 0,C 180,E1 -24772.804,E2 -24772.804} C_VEL
LIN {X 0,Y 140.793,Z 409.544,A -85,B 0,C 180,E1 -24776.04,E2 -24776.04} C_VEL
LIN {X 0,Y 138.658,Z 418.352,A -85,B 0,C 180,E1 -24779.433,E2 -24779.433} C_VEL
LIN {X 0,Y 136.548,Z 426.785,A -85,B 0,C 180,E1 -24783.476,E2 -24783.476} C_VEL
LIN {X 0,Y 135.13,Z 433.585,A -85,B 0,C 180,E1 -24787.572,E2 -24787.572} C_VEL
LIN {X 0,Y 134.119,Z 439.124,A -85,B 0,C 180,E1 -24791.732,E2 -24791.732} C_VEL
LIN {X 0,Y 133.389,Z 444.326,A -85,B 0,C 180,E1 -24796.77,E2 -24796.77} C_VEL
LIN {X 0,Y 133.301,Z 448.434,A -85,B 0,C 180,E1 -24802.256,E2 -24802.256} C_VEL
LIN {X 0,Y 134.047,Z 450.872,A -85,B 0,C 180,E1 -24807.011,E2 -24807.011} C_VEL
LIN {X 0,Y 135.731,Z 452.426,A -85,B 0,C 180,E1 -24812.226,E2 -24812.226} C_VEL
LIN {X 0,Y 137.909,Z 452.799,A -85,B 0,C 180,E1 -24816.521,E2 -24816.521} C_VEL
LIN {X 0,Y 141.122,Z 452.233,A -85,B 0,C 180,E1 -24821.106,E2 -24821.106} C_VEL
LIN {X 0,Y 145.663,Z 450.364,A -85,B 0,C 180,E1 -24826.041,E2 -24826.041} C_VEL
LIN {X 0,Y 151.631,Z 446.844,A -85,B 0,C 180,E1 -24830.901,E2 -24830.901} C_VEL
LIN {X 0,Y 157.863,Z 442.249,A -85,B 0,C 180,E1 -24834.893,E2 -24834.893} C_VEL
LIN {X 0,Y 163.857,Z 437.021,A -85,B 0,C 180,E1 -24838.157,E2 -24838.157} C_VEL
LIN {X 0,Y 170.966,Z 429.877,A -85,B 0,C 180,E1 -24841.378,E2 -24841.378} C_VEL
LIN {X 0,Y 178.352,Z 421.079,A -85,B 0,C 180,E1 -24844.221,E2 -24844.221} C_VEL
LIN {X 0,Y 185.216,Z 411.527,A -85,B 0,C 180,E1 -24846.537,E2 -24846.537} C_VEL
LIN {X 0,Y 191.51,Z 401.058,A -85,B 0,C 180,E1 -24848.442,E2 -24848.442} C_VEL
LIN {X 0,Y 197.169,Z 389.674,A -85,B 0,C 180,E1 -24850.008,E2 -24850.008} C_VEL
LIN {X 0,Y 201.776,Z 378.22,A -85,B 0,C 180,E1 -24851.195,E2 -24851.195} C_VEL
LIN {X 0,Y 205.434,Z 366.292,A -85,B 0,C 180,E1 -24852.152,E2 -24852.152} C_VEL
LIN {X 0,Y 208.536,Z 352.536,A -85,B 0,C 180,E1 -24852.898,E2 -24852.898} C_VEL
LIN {X 0,Y 210.851,Z 336.707,A -85,B 0,C 180,E1 -24853.493,E2 -24853.493} C_VEL
LIN {X 0,Y 209.451,Z 333.146,A -85,B 0,C 180,E1 -24855.686,E2 -24855.686} C_VEL
LIN {X 0,Y 207.913,Z 329.894,A -85,B 0,C 180,E1 -24858.85,E2 -24858.85} C_VEL
LIN {X 0,Y 206.994,Z 328.436,A -85,B 0,C 180,E1 -24861.931,E2 -24861.931} C_VEL
LIN {X 0,Y 206.683,Z 328.694,A -85,B 0,C 180,E1 -24865.725,E2 -24865.725} C_VEL
LIN {X 0,Y 206.984,Z 330.333,A -85,B 0,C 180,E1 -24868.506,E2 -24868.506} C_VEL
LIN {X 0,Y 208.09,Z 334.56,A -85,B 0,C 180,E1 -24872.077,E2 -24872.077} C_VEL
LIN {X 0,Y 209.171,Z 338.498,A -85,B 0,C 180,E1 -24874.285,E2 -24874.285} C_VEL
LIN {X 0,Y 210.176,Z 342.547,A -85,B 0,C 180,E1 -24876.088,E2 -24876.088} C_VEL
LIN {X 0,Y 207.288,Z 361.303,A -85,B 0,C 180,E1 -24876.814,E2 -24876.814} C_VEL
LIN {X 0,Y 204.126,Z 373.862,A -85,B 0,C 180,E1 -24877.424,E2 -24877.424} C_VEL
LIN {X 0,Y 199.47,Z 387.366,A -85,B 0,C 180,E1 -24878.385,E2 -24878.385} C_VEL
LIN {X 0,Y 194.6,Z 398.538,A -85,B 0,C 180,E1 -24879.477,E2 -24879.477} C_VEL
LIN {X 0,Y 189.139,Z 408.871,A -85,B 0,C 180,E1 -24880.799,E2 -24880.799} C_VEL
LIN {X 0,Y 183.224,Z 418.405,A -85,B 0,C 180,E1 -24882.413,E2 -24882.413} C_VEL
LIN {X 0,Y 175.758,Z 428.818,A -85,B 0,C 180,E1 -24884.79,E2 -24884.79} C_VEL
LIN {X 0,Y 168.686,Z 437.312,A -85,B 0,C 180,E1 -24887.394,E2 -24887.394} C_VEL
LIN {X 0,Y 161.07,Z 445.207,A -85,B 0,C 180,E1 -24890.757,E2 -24890.757} C_VEL
LIN {X 0,Y 155.159,Z 450.629,A -85,B 0,C 180,E1 -24893.929,E2 -24893.929} C_VEL
LIN {X 0,Y 149.854,Z 455.003,A -85,B 0,C 180,E1 -24897.365,E2 -24897.365} C_VEL
LIN {X 0,Y 145.281,Z 458.387,A -85,B 0,C 180,E1 -24901.073,E2 -24901.073} C_VEL
LIN {X 0,Y 140.15,Z 461.507,A -85,B 0,C 180,E1 -24906.396,E2 -24906.396} C_VEL
LIN {X 0,Y 136.443,Z 463.111,A -85,B 0,C 180,E1 -24912,E2 -24912} C_VEL
LIN {X 0,Y 134.401,Z 463.221,A -85,B 0,C 180,E1 -24917.928,E2 -24917.928} C_VEL
LIN {X 0,Y 134.175,Z 463.048,A -85,B 0,C 180,E1 -24918.997,E2 -24918.997} C_VEL
LIN {X 0,Y 133.187,Z 462.561,A -85,B 0,C 180,E1 -24921.481,E2 -24921.481} C_VEL
LIN {X 0,Y 131.52,Z 461.656,A -85,B 0,C 180,E1 -24923.92,E2 -24923.92} C_VEL
LIN {X 0,Y 127.986,Z 458.862,A -85,B 0,C 180,E1 -24928.841,E2 -24928.841} C_VEL
LIN {X 0,Y 126.982,Z 456.396,A -85,B 0,C 180,E1 -24932.238,E2 -24932.238} C_VEL
LIN {X 0,Y 126.94,Z 452.778,A -85,B 0,C 180,E1 -24936.356,E2 -24936.356} C_VEL
LIN {X 0,Y 127.539,Z 446.358,A -85,B 0,C 180,E1 -24941.924,E2 -24941.924} C_VEL
LIN {X 0,Y 128.779,Z 439.26,A -85,B 0,C 180,E1 -24946.647,E2 -24946.647} C_VEL
LIN {X 0,Y 130.805,Z 430.337,A -85,B 0,C 180,E1 -24951.261,E2 -24951.261} C_VEL
LIN {X 0,Y 133.088,Z 421.194,A -85,B 0,C 180,E1 -24954.987,E2 -24954.987} C_VEL
LIN {X 0,Y 135.472,Z 411.48,A -85,B 0,C 180,E1 -24958.122,E2 -24958.122} C_VEL
LIN {X 0,Y 137.819,Z 401.543,A -85,B 0,C 180,E1 -24960.656,E2 -24960.656} C_VEL
LIN {X 0,Y 140.397,Z 389.717,A -85,B 0,C 180,E1 -24962.978,E2 -24962.978} C_VEL
LIN {X 0,Y 142.517,Z 377.66,A -85,B 0,C 180,E1 -24964.758,E2 -24964.758} C_VEL
LIN {X 0,Y 144.393,Z 363.808,A -85,B 0,C 180,E1 -24966.163,E2 -24966.163} C_VEL
LIN {X 0,Y 146.035,Z 342.22,A -85,B 0,C 180,E1 -24967.518,E2 -24967.518} C_VEL
LIN {X 0,Y 147.65,Z 317.758,A -85,B 0,C 180,E1 -24968.929,E2 -24968.929} C_VEL
LIN {X 0,Y 145.881,Z 297.73,A -85,B 0,C 180,E1 -24970.642,E2 -24970.642} C_VEL
LIN {X 0,Y 139.724,Z 278.891,A -85,B 0,C 180,E1 -24973.299,E2 -24973.299} C_VEL
LIN {X 0,Y 133.484,Z 263.082,A -85,B 0,C 180,E1 -24975.991,E2 -24975.991} C_VEL
LIN {X 0,Y 130.116,Z 256.561,A -85,B 0,C 180,E1 -24977.4,E2 -24977.4} C_VEL
LIN {X 0,Y 128.936,Z 253.426,A -85,B 0,C 180,E1 -24978.042,E2 -24978.042} C_VEL
LIN {X 0,Y 128.945,Z 253.417,A -85,B 0,C 180,E1 -24984.831,E2 -24984.831} C_VEL
LIN {X 0,Y 129.007,Z 253.416,A -85,B 0,C 180,E1 -24990.638,E2 -24990.638} C_VEL
LIN {X 0,Y 129.056,Z 253.41,A -85,B 0,C 180,E1 -24997.768,E2 -24997.768} C_VEL
LIN {X 0,Y 129.131,Z 253.374,A -85,B 0,C 180,E1 -25004.208,E2 -25004.208} C_VEL
LIN {X 0,Y 129.328,Z 253.37,A -85,B 0,C 180,E1 -25007.972,E2 -25007.972} C_VEL
LIN {X 0,Y 129.444,Z 253.361,A -85,B 0,C 180,E1 -25010.625,E2 -25010.625} C_VEL
LIN {X 0,Y 130.053,Z 253.246,A -85,B 0,C 180,E1 -25019.999,E2 -25019.999} C_VEL
LIN {X 0,Y 129.444,Z 253.359,A -85,B 0,C 180,E1 -25029.373,E2 -25029.373} C_VEL
LIN {X 0,Y 129.285,Z 253.368,A -85,B 0,C 180,E1 -25032.558,E2 -25032.558} C_VEL
LIN {X 0,Y 129.129,Z 253.347,A -85,B 0,C 180,E1 -25039.059,E2 -25039.059} C_VEL
LIN {X 0,Y 129.098,Z 253.376,A -85,B 0,C 180,E1 -25042.399,E2 -25042.399} C_VEL
LIN {X 0,Y 129.02,Z 253.406,A -85,B 0,C 180,E1 -25045.834,E2 -25045.834} C_VEL
LIN {X 0,Y 129.004,Z 253.415,A -85,B 0,C 180,E1 -25049.36,E2 -25049.36} C_VEL
LIN {X 0,Y 128.98,Z 253.398,A -85,B 0,C 180,E1 -25055.19,E2 -25055.19} C_VEL
LIN {X 0,Y 128.97,Z 253.375,A -85,B 0,C 180,E1 -25060.836,E2 -25060.836} C_VEL
LIN {X 0,Y 128.916,Z 253.416,A -85,B 0,C 180,E1 -25065.128,E2 -25065.128} C_VEL
LIN {X 0,Y 128.934,Z 253.425,A -85,B 0,C 180,E1 -25069.738,E2 -25069.738} C_VEL
LIN {X 0,Y 128.951,Z 253.402,A -85,B 0,C 180,E1 -25074.835,E2 -25074.835} C_VEL
LIN {X 0,Y 129.011,Z 253.398,A -85,B 0,C 180,E1 -25080.645,E2 -25080.645} C_VEL
LIN {X 0,Y 129.025,Z 253.414,A -85,B 0,C 180,E1 -25084.17,E2 -25084.17} C_VEL
LIN {X 0,Y 129.103,Z 253.398,A -85,B 0,C 180,E1 -25087.73,E2 -25087.73} C_VEL
LIN {X 0,Y 129.156,Z 253.376,A -85,B 0,C 180,E1 -25090.947,E2 -25090.947} C_VEL
LIN {X 0,Y 129.414,Z 253.362,A -85,B 0,C 180,E1 -25097.822,E2 -25097.822} C_VEL
LIN {X 0,Y 129.512,Z 253.34,A -85,B 0,C 180,E1 -25100.632,E2 -25100.632} C_VEL
LIN {X 0,Y 130.088,Z 253.282,A -85,B 0,C 180,E1 -25110,E2 -25110} C_VEL
LIN {X 0,Y 129.678,Z 253.33,A -85,B 0,C 180,E1 -25113.194,E2 -25113.194} C_VEL
LIN {X 0,Y 130.627,Z 256.184,A -85,B 0,C 180,E1 -25113.692,E2 -25113.692} C_VEL
LIN {X 0,Y 136.985,Z 268.679,A -85,B 0,C 180,E1 -25116.281,E2 -25116.281} C_VEL
LIN {X 0,Y 145.237,Z 288.046,A -85,B 0,C 180,E1 -25119.509,E2 -25119.509} C_VEL
LIN {X 0,Y 148.733,Z 297.015,A -85,B 0,C 180,E1 -25120.811,E2 -25120.811} C_VEL
LIN {X 0,Y 144.735,Z 349.258,A -85,B 0,C 180,E1 -25123.8,E2 -25123.8} C_VEL
LIN {X 0,Y 143.314,Z 362.528,A -85,B 0,C 180,E1 -25125.099,E2 -25125.099} C_VEL
LIN {X 0,Y 141.455,Z 374.726,A -85,B 0,C 180,E1 -25126.784,E2 -25126.784} C_VEL
LIN {X 0,Y 139.224,Z 386.186,A -85,B 0,C 180,E1 -25128.902,E2 -25128.902} C_VEL
LIN {X 0,Y 136.881,Z 397.065,A -85,B 0,C 180,E1 -25131.51,E2 -25131.51} C_VEL
LIN {X 0,Y 134.323,Z 407.698,A -85,B 0,C 180,E1 -25134.742,E2 -25134.742} C_VEL
LIN {X 0,Y 131.81,Z 417.767,A -85,B 0,C 180,E1 -25138.674,E2 -25138.674} C_VEL
LIN {X 0,Y 129.635,Z 426.179,A -85,B 0,C 180,E1 -25142.826,E2 -25142.826} C_VEL
LIN {X 0,Y 128.13,Z 433.076,A -85,B 0,C 180,E1 -25147.106,E2 -25147.106} C_VEL
LIN {X 0,Y 127.033,Z 438.867,A -85,B 0,C 180,E1 -25151.592,E2 -25151.592} C_VEL
LIN {X 0,Y 126.335,Z 443.681,A -85,B 0,C 180,E1 -25156.312,E2 -25156.312} C_VEL
LIN {X 0,Y 126.198,Z 448.178,A -85,B 0,C 180,E1 -25162.224,E2 -25162.224} C_VEL
LIN {X 0,Y 126.779,Z 450.423,A -85,B 0,C 180,E1 -25166.335,E2 -25166.335} C_VEL
LIN {X 0,Y 128.181,Z 452.249,A -85,B 0,C 180,E1 -25171.302,E2 -25171.302} C_VEL
LIN {X 0,Y 130.485,Z 453.114,A -85,B 0,C 180,E1 -25176.281,E2 -25176.281} C_VEL
LIN {X 0,Y 134.129,Z 452.907,A -85,B 0,C 180,E1 -25181.677,E2 -25181.677} C_VEL
LIN {X 0,Y 137.757,Z 451.798,A -85,B 0,C 180,E1 -25185.748,E2 -25185.748} C_VEL
LIN {X 0,Y 142.67,Z 449.554,A -85,B 0,C 180,E1 -25190.099,E2 -25190.099} C_VEL
LIN {X 0,Y 149.188,Z 445.708,A -85,B 0,C 180,E1 -25194.595,E2 -25194.595} C_VEL
LIN {X 0,Y 156.871,Z 439.945,A -85,B 0,C 180,E1 -25198.908,E2 -25198.908} C_VEL
LIN {X 0,Y 163.119,Z 434.409,A -85,B 0,C 180,E1 -25201.817,E2 -25201.817} C_VEL
LIN {X 0,Y 170.555,Z 426.885,A -85,B 0,C 180,E1 -25204.728,E2 -25204.728} C_VEL
LIN {X 0,Y 177.763,Z 418.214,A -85,B 0,C 180,E1 -25207.203,E2 -25207.203} C_VEL
LIN {X 0,Y 185.218,Z 407.589,A -85,B 0,C 180,E1 -25209.442,E2 -25209.442} C_VEL
LIN {X 0,Y 191.622,Z 396.424,A -85,B 0,C 180,E1 -25211.179,E2 -25211.179} C_VEL
LIN {X 0,Y 196.528,Z 386.21,A -85,B 0,C 180,E1 -25212.391,E2 -25212.391} C_VEL
LIN {X 0,Y 201.218,Z 373.951,A -85,B 0,C 180,E1 -25213.548,E2 -25213.548} C_VEL
LIN {X 0,Y 204.924,Z 360.959,A -85,B 0,C 180,E1 -25214.401,E2 -25214.401} C_VEL
LIN {X 0,Y 207.511,Z 347.832,A -85,B 0,C 180,E1 -25214.969,E2 -25214.969} C_VEL
LIN {X 0,Y 208.442,Z 341.236,A -85,B 0,C 180,E1 -25215.228,E2 -25215.228} C_VEL
LIN {X 0,Y 207.495,Z 339.147,A -85,B 0,C 180,E1 -25216.866,E2 -25216.866} C_VEL
LIN {X 0,Y 206.529,Z 336.707,A -85,B 0,C 180,E1 -25219.281,E2 -25219.281} C_VEL
LIN {X 0,Y 205.777,Z 335.421,A -85,B 0,C 180,E1 -25222.068,E2 -25222.068} C_VEL
LIN {X 0,Y 205.5,Z 335.782,A -85,B 0,C 180,E1 -25225.884,E2 -25225.884} C_VEL
LIN {X 0,Y 205.691,Z 337.139,A -85,B 0,C 180,E1 -25228.042,E2 -25228.042} C_VEL
LIN {X 0,Y 206.57,Z 341.078,A -85,B 0,C 180,E1 -25231.411,E2 -25231.411} C_VEL
LIN {X 0,Y 207.309,Z 344.339,A -85,B 0,C 180,E1 -25233.284,E2 -25233.284} C_VEL
LIN {X 0,Y 207.835,Z 346.537,A -85,B 0,C 180,E1 -25234.352,E2 -25234.352} C_VEL
LIN {X 0,Y 205.255,Z 361.719,A -85,B 0,C 180,E1 -25234.922,E2 -25234.922} C_VEL
LIN {X 0,Y 201.591,Z 375.176,A -85,B 0,C 180,E1 -25235.577,E2 -25235.577} C_VEL
LIN {X 0,Y 196.739,Z 388.4,A -85,B 0,C 180,E1 -25236.518,E2 -25236.518} C_VEL
LIN {X 0,Y 190.289,Z 401.917,A -85,B 0,C 180,E1 -25237.874,E2 -25237.874} C_VEL
LIN {X 0,Y 184.002,Z 412.725,A -85,B 0,C 180,E1 -25239.343,E2 -25239.343} C_VEL
LIN {X 0,Y 177.316,Z 422.436,A -85,B 0,C 180,E1 -25241.15,E2 -25241.15} C_VEL
LIN {X 0,Y 169.677,Z 431.954,A -85,B 0,C 180,E1 -25243.55,E2 -25243.55} C_VEL
LIN {X 0,Y 162.431,Z 439.746,A -85,B 0,C 180,E1 -25246.195,E2 -25246.195} C_VEL
LIN {X 0,Y 155.692,Z 446.143,A -85,B 0,C 180,E1 -25249.121,E2 -25249.121} C_VEL
LIN {X 0,Y 149.516,Z 451.319,A -85,B 0,C 180,E1 -25252.338,E2 -25252.338} C_VEL
LIN {X 0,Y 143.946,Z 455.423,A -85,B 0,C 180,E1 -25255.846,E2 -25255.846} C_VEL
LIN {X 0,Y 139.104,Z 458.582,A -85,B 0,C 180,E1 -25259.657,E2 -25259.657} C_VEL
LIN {X 0,Y 133.681,Z 461.468,A -85,B 0,C 180,E1 -25265.131,E2 -25265.131} C_VEL
LIN {X 0,Y 129.682,Z 462.818,A -85,B 0,C 180,E1 -25271.026,E2 -25271.026} C_VEL
LIN {X 0,Y 127.461,Z 462.752,A -85,B 0,C 180,E1 -25277.26,E2 -25277.26} C_VEL
LIN {X 0,Y 126.682,Z 461.18,A -85,B 0,C 180,E1 -25283.63,E2 -25283.63} C_VEL
LIN {X 0,Y 126.79,Z 459.8,A -85,B 0,C 180,E1 -25286.823,E2 -25286.823} C_VEL
LIN {X 0,Y 127.013,Z 457.995,A -85,B 0,C 180,E1 -25290,E2 -25290} C_VEL
LIN {X 0,Y 126.982,Z 456.396,A -85,B 0,C 180,E1 -25292.238,E2 -25292.238} C_VEL
LIN {X 0,Y 126.343,Z 454.279,A -85,B 0,C 180,E1 -25294.708,E2 -25294.708} C_VEL
LIN {X 0,Y 124.838,Z 451.818,A -85,B 0,C 180,E1 -25297.083,E2 -25297.083} C_VEL
LIN {X 0,Y 121.241,Z 445.045,A -85,B 0,C 180,E1 -25302.547,E2 -25302.547} C_VEL
LIN {X 0,Y 121.091,Z 441.729,A -85,B 0,C 180,E1 -25304.896,E2 -25304.896} C_VEL
LIN {X 0,Y 123.002,Z 433.166,A -85,B 0,C 180,E1 -25310.046,E2 -25310.046} C_VEL
LIN {X 0,Y 125.057,Z 424.718,A -85,B 0,C 180,E1 -25314.041,E2 -25314.041} C_VEL
LIN {X 0,Y 127.572,Z 415.227,A -85,B 0,C 180,E1 -25317.575,E2 -25317.575} C_VEL
LIN {X 0,Y 130.383,Z 404.111,A -85,B 0,C 180,E1 -25320.796,E2 -25320.796} C_VEL
LIN {X 0,Y 132.937,Z 393.079,A -85,B 0,C 180,E1 -25323.259,E2 -25323.259} C_VEL
LIN {X 0,Y 135.287,Z 380.933,A -85,B 0,C 180,E1 -25325.3,E2 -25325.3} C_VEL
LIN {X 0,Y 137.374,Z 367.038,A -85,B 0,C 180,E1 -25326.945,E2 -25326.945} C_VEL
LIN {X 0,Y 138.688,Z 354.127,A -85,B 0,C 180,E1 -25327.926,E2 -25327.926} C_VEL
LIN {X 0,Y 141.198,Z 318.372,A -85,B 0,C 180,E1 -25330.067,E2 -25330.067} C_VEL
LIN {X 0,Y 139.639,Z 299.809,A -85,B 0,C 180,E1 -25331.745,E2 -25331.745} C_VEL
LIN {X 0,Y 133.868,Z 281.941,A -85,B 0,C 180,E1 -25334.393,E2 -25334.393} C_VEL
LIN {X 0,Y 127.902,Z 266.527,A -85,B 0,C 180,E1 -25337.156,E2 -25337.156} C_VEL
LIN {X 0,Y 123.204,Z 257.616,A -85,B 0,C 180,E1 -25339.283,E2 -25339.283} C_VEL
LIN {X 0,Y 121.988,Z 254.955,A -85,B 0,C 180,E1 -25339.89,E2 -25339.89} C_VEL
LIN {X 0,Y 121.857,Z 254.308,A -85,B 0,C 180,E1 -25340.063,E2 -25340.063} C_VEL
LIN {X 0,Y 121.897,Z 254.295,A -85,B 0,C 180,E1 -25344.79,E2 -25344.79} C_VEL
LIN {X 0,Y 121.916,Z 254.3,A -85,B 0,C 180,E1 -25349.836,E2 -25349.836} C_VEL
LIN {X 0,Y 121.974,Z 254.29,A -85,B 0,C 180,E1 -25357.19,E2 -25357.19} C_VEL
LIN {X 0,Y 122.045,Z 254.258,A -85,B 0,C 180,E1 -25363.265,E2 -25363.265} C_VEL
LIN {X 0,Y 122.272,Z 254.247,A -85,B 0,C 180,E1 -25367.693,E2 -25367.693} C_VEL
LIN {X 0,Y 122.39,Z 254.234,A -85,B 0,C 180,E1 -25373.404,E2 -25373.404} C_VEL
LIN {X 0,Y 123.007,Z 254.123,A -85,B 0,C 180,E1 -25379.999,E2 -25379.999} C_VEL
LIN {X 0,Y 122.362,Z 254.237,A -85,B 0,C 180,E1 -25387.108,E2 -25387.108} C_VEL
LIN {X 0,Y 122.273,Z 254.242,A -85,B 0,C 180,E1 -25392.308,E2 -25392.308} C_VEL
LIN {X 0,Y 122.079,Z 254.232,A -85,B 0,C 180,E1 -25396.728,E2 -25396.728} C_VEL
LIN {X 0,Y 122.017,Z 254.259,A -85,B 0,C 180,E1 -25402.858,E2 -25402.858} C_VEL
LIN {X 0,Y 121.93,Z 254.294,A -85,B 0,C 180,E1 -25407.458,E2 -25407.458} C_VEL
LIN {X 0,Y 121.895,Z 254.298,A -85,B 0,C 180,E1 -25411.257,E2 -25411.257} C_VEL
LIN {X 0,Y 121.901,Z 254.272,A -85,B 0,C 180,E1 -25416.191,E2 -25416.191} C_VEL
LIN {X 0,Y 121.896,Z 254.259,A -85,B 0,C 180,E1 -25421.459,E2 -25421.459} C_VEL
LIN {X 0,Y 121.864,Z 254.305,A -85,B 0,C 180,E1 -25428.564,E2 -25428.564} C_VEL
LIN {X 0,Y 121.903,Z 254.279,A -85,B 0,C 180,E1 -25434.798,E2 -25434.798} C_VEL
LIN {X 0,Y 121.921,Z 254.275,A -85,B 0,C 180,E1 -25439.842,E2 -25439.842} C_VEL
LIN {X 0,Y 121.979,Z 254.29,A -85,B 0,C 180,E1 -25446.218,E2 -25446.218} C_VEL
LIN {X 0,Y 122.045,Z 254.265,A -85,B 0,C 180,E1 -25449.79,E2 -25449.79} C_VEL
LIN {X 0,Y 122.261,Z 254.255,A -85,B 0,C 180,E1 -25456.709,E2 -25456.709} C_VEL
LIN {X 0,Y 122.442,Z 254.22,A -85,B 0,C 180,E1 -25460.086,E2 -25460.086} C_VEL
LIN {X 0,Y 122.604,Z 254.208,A -85,B 0,C 180,E1 -25466.714,E2 -25466.714} C_VEL
LIN {X 0,Y 123.042,Z 254.16,A -85,B 0,C 180,E1 -25470,E2 -25470} C_VEL
LIN {X 0,Y 122.843,Z 254.182,A -85,B 0,C 180,E1 -25471.24,E2 -25471.24} C_VEL
LIN {X 0,Y 123.858,Z 257.206,A -85,B 0,C 180,E1 -25471.857,E2 -25471.857} C_VEL
LIN {X 0,Y 131.506,Z 272.571,A -85,B 0,C 180,E1 -25475.27,E2 -25475.27} C_VEL
LIN {X 0,Y 139.294,Z 291.007,A -85,B 0,C 180,E1 -25478.484,E2 -25478.484} C_VEL
LIN {X 0,Y 142.27,Z 298.749,A -85,B 0,C 180,E1 -25479.682,E2 -25479.682} C_VEL
LIN {X 0,Y 138.186,Z 349.662,A -85,B 0,C 180,E1 -25482.704,E2 -25482.704} C_VEL
LIN {X 0,Y 136.618,Z 363.452,A -85,B 0,C 180,E1 -25484.118,E2 -25484.118} C_VEL
LIN {X 0,Y 134.654,Z 375.639,A -85,B 0,C 180,E1 -25485.902,E2 -25485.902} C_VEL
LIN {X 0,Y 132.138,Z 387.983,A -85,B 0,C 180,E1 -25488.354,E2 -25488.354} C_VEL
LIN {X 0,Y 129.387,Z 399.992,A -85,B 0,C 180,E1 -25491.507,E2 -25491.507} C_VEL
LIN {X 0,Y 126.765,Z 410.258,A -85,B 0,C 180,E1 -25495.005,E2 -25495.005} C_VEL
LIN {X 0,Y 124.224,Z 419.963,A -85,B 0,C 180,E1 -25499.202,E2 -25499.202} C_VEL
LIN {X 0,Y 121.899,Z 428.967,A -85,B 0,C 180,E1 -25504.219,E2 -25504.219} C_VEL
LIN {X 0,Y 120.467,Z 435.882,A -85,B 0,C 180,E1 -25509.152,E2 -25509.152} C_VEL
LIN {X 0,Y 119.387,Z 442.307,A -85,B 0,C 180,E1 -25515.058,E2 -25515.058} C_VEL
LIN {X 0,Y 119.034,Z 446.477,A -85,B 0,C 180,E1 -25520.127,E2 -25520.127} C_VEL
LIN {X 0,Y 119.476,Z 449.731,A -85,B 0,C 180,E1 -25525.431,E2 -25525.431} C_VEL
LIN {X 0,Y 120.805,Z 451.988,A -85,B 0,C 180,E1 -25530.757,E2 -25530.757} C_VEL
LIN {X 0,Y 123.282,Z 453.335,A -85,B 0,C 180,E1 -25536.482,E2 -25536.482} C_VEL
LIN {X 0,Y 126.249,Z 453.547,A -85,B 0,C 180,E1 -25541.129,E2 -25541.129} C_VEL
LIN {X 0,Y 130.364,Z 452.809,A -85,B 0,C 180,E1 -25545.998,E2 -25545.998} C_VEL
LIN {X 0,Y 135.985,Z 450.769,A -85,B 0,C 180,E1 -25551.082,E2 -25551.082} C_VEL
LIN {X 0,Y 143.185,Z 447.03,A -85,B 0,C 180,E1 -25555.997,E2 -25555.997} C_VEL
LIN {X 0,Y 150.44,Z 442.254,A -85,B 0,C 180,E1 -25560.001,E2 -25560.001} C_VEL
LIN {X 0,Y 157.389,Z 436.805,A -85,B 0,C 180,E1 -25563.201,E2 -25563.201} C_VEL
LIN {X 0,Y 165.152,Z 429.621,A -85,B 0,C 180,E1 -25566.192,E2 -25566.192} C_VEL
LIN {X 0,Y 173.493,Z 420.457,A -85,B 0,C 180,E1 -25568.931,E2 -25568.931} C_VEL
LIN {X 0,Y 180.459,Z 411.404,A -85,B 0,C 180,E1 -25570.927,E2 -25570.927} C_VEL
LIN {X 0,Y 187.298,Z 400.745,A -85,B 0,C 180,E1 -25572.71,E2 -25572.71} C_VEL
LIN {X 0,Y 192.65,Z 390.714,A -85,B 0,C 180,E1 -25573.987,E2 -25573.987} C_VEL
LIN {X 0,Y 197.655,Z 379.223,A -85,B 0,C 180,E1 -25575.103,E2 -25575.103} C_VEL
LIN {X 0,Y 201.817,Z 366.606,A -85,B 0,C 180,E1 -25576.046,E2 -25576.046} C_VEL
LIN {X 0,Y 204.942,Z 353.687,A -85,B 0,C 180,E1 -25576.687,E2 -25576.687} C_VEL
LIN {X 0,Y 206.206,Z 346.202,A -85,B 0,C 180,E1 -25576.985,E2 -25576.985} C_VEL
LIN {X 0,Y 205.1,Z 343.405,A -85,B 0,C 180,E1 -25579.885,E2 -25579.885} C_VEL
LIN {X 0,Y 204.563,Z 342.406,A -85,B 0,C 180,E1 -25582.206,E2 -25582.206} C_VEL
LIN {X 0,Y 204.29,Z 342.721,A -85,B 0,C 180,E1 -25585.603,E2 -25585.603} C_VEL
LIN {X 0,Y 204.419,Z 343.822,A -85,B 0,C 180,E1 -25587.483,E2 -25587.483} C_VEL
LIN {X 0,Y 205.086,Z 347.664,A -85,B 0,C 180,E1 -25590.774,E2 -25590.774} C_VEL
LIN {X 0,Y 205.632,Z 350.742,A -85,B 0,C 180,E1 -25592.557,E2 -25592.557} C_VEL
LIN {X 0,Y 202.707,Z 365.295,A -85,B 0,C 180,E1 -25593.148,E2 -25593.148} C_VEL
LIN {X 0,Y 198.756,Z 378.28,A -85,B 0,C 180,E1 -25593.795,E2 -25593.795} C_VEL
LIN {X 0,Y 193.501,Z 391.213,A -85,B 0,C 180,E1 -25594.749,E2 -25594.749} C_VEL
LIN {X 0,Y 187.599,Z 402.786,A -85,B 0,C 180,E1 -25595.899,E2 -25595.899} C_VEL
LIN {X 0,Y 180.412,Z 414.255,A -85,B 0,C 180,E1 -25597.474,E2 -25597.474} C_VEL
LIN {X 0,Y 172.841,Z 424.467,A -85,B 0,C 180,E1 -25599.422,E2 -25599.422} C_VEL
LIN {X 0,Y 164.953,Z 433.547,A -85,B 0,C 180,E1 -25601.796,E2 -25601.796} C_VEL
LIN {X 0,Y 157.468,Z 440.944,A -85,B 0,C 180,E1 -25604.437,E2 -25604.437} C_VEL
LIN {X 0,Y 150.45,Z 446.989,A -85,B 0,C 180,E1 -25607.369,E2 -25607.369} C_VEL
LIN {X 0,Y 143.979,Z 451.908,A -85,B 0,C 180,E1 -25610.617,E2 -25610.617} C_VEL
LIN {X 0,Y 138.129,Z 455.813,A -85,B 0,C 180,E1 -25614.193,E2 -25614.193} C_VEL
LIN {X 0,Y 133.018,Z 458.785,A -85,B 0,C 180,E1 -25618.11,E2 -25618.11} C_VEL
LIN {X 0,Y 127.249,Z 461.371,A -85,B 0,C 180,E1 -25623.781,E2 -25623.781} C_VEL
LIN {X 0,Y 122.968,Z 462.529,A -85,B 0,C 180,E1 -25629.947,E2 -25629.947} C_VEL
LIN {X 0,Y 120.546,Z 462.232,A -85,B 0,C 180,E1 -25636.515,E2 -25636.515} C_VEL
LIN {X 0,Y 119.647,Z 460.443,A -85,B 0,C 180,E1 -25643.254,E2 -25643.254} C_VEL
LIN {X 0,Y 119.725,Z 458.97,A -85,B 0,C 180,E1 -25646.635,E2 -25646.635} C_VEL
LIN {X 0,Y 119.962,Z 457.063,A -85,B 0,C 180,E1 -25650,E2 -25650} C_VEL
LIN {X 0,Y 119.911,Z 453.309,A -85,B 0,C 180,E1 -25654.87,E2 -25654.87} C_VEL
LIN {X 0,Y 120.297,Z 446.966,A -85,B 0,C 180,E1 -25660.944,E2 -25660.944} C_VEL
LIN {X 0,Y 121.091,Z 441.729,A -85,B 0,C 180,E1 -25664.896,E2 -25664.896} C_VEL
LIN {X 0,Y 121.113,Z 438.263,A -85,B 0,C 180,E1 -25667.138,E2 -25667.138} C_VEL
LIN {X 0,Y 119.679,Z 432.007,A -85,B 0,C 180,E1 -25670.717,E2 -25670.717} C_VEL
LIN {X 0,Y 118.565,Z 425.133,A -85,B 0,C 180,E1 -25674.155,E2 -25674.155} C_VEL
LIN {X 0,Y 119.102,Z 420.705,A -85,B 0,C 180,E1 -25676.085,E2 -25676.085} C_VEL
LIN {X 0,Y 121.908,Z 410.125,A -85,B 0,C 180,E1 -25679.846,E2 -25679.846} C_VEL
LIN {X 0,Y 124.679,Z 399.115,A -85,B 0,C 180,E1 -25682.853,E2 -25682.853} C_VEL
LIN {X 0,Y 127.511,Z 386.955,A -85,B 0,C 180,E1 -25685.356,E2 -25685.356} C_VEL
LIN {X 0,Y 129.814,Z 374.112,A -85,B 0,C 180,E1 -25687.272,E2 -25687.272} C_VEL
LIN {X 0,Y 131.555,Z 360.931,A -85,B 0,C 180,E1 -25688.631,E2 -25688.631} C_VEL
LIN {X 0,Y 134.771,Z 318.818,A -85,B 0,C 180,E1 -25691.331,E2 -25691.331} C_VEL
LIN {X 0,Y 133.366,Z 301.578,A -85,B 0,C 180,E1 -25692.959,E2 -25692.959} C_VEL
LIN {X 0,Y 127.02,Z 281.979,A -85,B 0,C 180,E1 -25696.077,E2 -25696.077} C_VEL
LIN {X 0,Y 121.413,Z 268.009,A -85,B 0,C 180,E1 -25698.885,E2 -25698.885} C_VEL
LIN {X 0,Y 116.357,Z 258.808,A -85,B 0,C 180,E1 -25701.333,E2 -25701.333} C_VEL
LIN {X 0,Y 114.991,Z 256.251,A -85,B 0,C 180,E1 -25702.047,E2 -25702.047} C_VEL
LIN {X 0,Y 114.784,Z 255.187,A -85,B 0,C 180,E1 -25702.244,E2 -25702.244} C_VEL
LIN {X 0,Y 114.844,Z 255.181,A -85,B 0,C 180,E1 -25708.941,E2 -25708.941} C_VEL
LIN {X 0,Y 114.895,Z 255.171,A -85,B 0,C 180,E1 -25716.553,E2 -25716.553} C_VEL
LIN {X 0,Y 114.95,Z 255.148,A -85,B 0,C 180,E1 -25722.199,E2 -25722.199} C_VEL
LIN {X 0,Y 115.289,Z 255.123,A -85,B 0,C 180,E1 -25729.461,E2 -25729.461} C_VEL
LIN {X 0,Y 115.471,Z 255.073,A -85,B 0,C 180,E1 -25736.509,E2 -25736.509} C_VEL
LIN {X 0,Y 115.934,Z 255.002,A -85,B 0,C 180,E1 -25739.999,E2 -25739.999} C_VEL
LIN {X 0,Y 115.334,Z 255.117,A -85,B 0,C 180,E1 -25746.999,E2 -25746.999} C_VEL
LIN {X 0,Y 115.192,Z 255.122,A -85,B 0,C 180,E1 -25752.561,E2 -25752.561} C_VEL
LIN {X 0,Y 114.987,Z 255.106,A -85,B 0,C 180,E1 -25757.793,E2 -25757.793} C_VEL
LIN {X 0,Y 114.937,Z 255.144,A -85,B 0,C 180,E1 -25763.495,E2 -25763.495} C_VEL
LIN {X 0,Y 114.851,Z 255.176,A -85,B 0,C 180,E1 -25771.064,E2 -25771.064} C_VEL
LIN {X 0,Y 114.801,Z 255.139,A -85,B 0,C 180,E1 -25777.747,E2 -25777.747} C_VEL
LIN {X 0,Y 114.8,Z 255.153,A -85,B 0,C 180,E1 -25782.731,E2 -25782.731} C_VEL
LIN {X 0,Y 114.787,Z 255.184,A -85,B 0,C 180,E1 -25787.669,E2 -25787.669} C_VEL
LIN {X 0,Y 114.78,Z 255.18,A -85,B 0,C 180,E1 -25792.747,E2 -25792.747} C_VEL
LIN {X 0,Y 114.85,Z 255.146,A -85,B 0,C 180,E1 -25798.946,E2 -25798.946} C_VEL
LIN {X 0,Y 114.944,Z 255.166,A -85,B 0,C 180,E1 -25806.509,E2 -25806.509} C_VEL
LIN {X 0,Y 115.014,Z 255.138,A -85,B 0,C 180,E1 -25812.212,E2 -25812.212} C_VEL
LIN {X 0,Y 115.282,Z 255.124,A -85,B 0,C 180,E1 -25817.265,E2 -25817.265} C_VEL
LIN {X 0,Y 115.385,Z 255.111,A -85,B 0,C 180,E1 -25823.004,E2 -25823.004} C_VEL
LIN {X 0,Y 115.841,Z 255.175,A -85,B 0,C 180,E1 -25829.131,E2 -25829.131} C_VEL
LIN {X 0,Y 117.056,Z 258.025,A -85,B 0,C 180,E1 -25829.818,E2 -25829.818} C_VEL
LIN {X 0,Y 126.08,Z 276.418,A -85,B 0,C 180,E1 -25834.17,E2 -25834.17} C_VEL
LIN {X 0,Y 133.531,Z 294.403,A -85,B 0,C 180,E1 -25837.498,E2 -25837.498} C_VEL
LIN {X 0,Y 135.818,Z 300.258,A -85,B 0,C 180,E1 -25838.453,E2 -25838.453} C_VEL
LIN {X 0,Y 131.638,Z 349.95,A -85,B 0,C 180,E1 -25841.536,E2 -25841.536} C_VEL
LIN {X 0,Y 129.876,Z 364.387,A -85,B 0,C 180,E1 -25843.09,E2 -25843.09} C_VEL
LIN {X 0,Y 127.758,Z 376.938,A -85,B 0,C 180,E1 -25845.069,E2 -25845.069} C_VEL
LIN {X 0,Y 124.882,Z 390.126,A -85,B 0,C 180,E1 -25847.878,E2 -25847.878} C_VEL
LIN {X 0,Y 122.197,Z 401.284,A -85,B 0,C 180,E1 -25851.071,E2 -25851.071} C_VEL
LIN {X 0,Y 119.439,Z 411.691,A -85,B 0,C 180,E1 -25854.888,E2 -25854.888} C_VEL
LIN {X 0,Y 116.804,Z 421.347,A -85,B 0,C 180,E1 -25859.417,E2 -25859.417} C_VEL
LIN {X 0,Y 114.728,Z 429.29,A -85,B 0,C 180,E1 -25864.183,E2 -25864.183} C_VEL
LIN {X 0,Y 113.153,Z 436.813,A -85,B 0,C 180,E1 -25869.937,E2 -25869.937} C_VEL
LIN {X 0,Y 112.301,Z 441.897,A -85,B 0,C 180,E1 -25874.931,E2 -25874.931} C_VEL
LIN {X 0,Y 111.953,Z 446.777,A -85,B 0,C 180,E1 -25881.116,E2 -25881.116} C_VEL
LIN {X 0,Y 112.889,Z 450.637,A -85,B 0,C 180,E1 -25888.054,E2 -25888.054} C_VEL
LIN {X 0,Y 115.127,Z 452.974,A -85,B 0,C 180,E1 -25894.704,E2 -25894.704} C_VEL
LIN {X 0,Y 118.808,Z 453.937,A -85,B 0,C 180,E1 -25901.15,E2 -25901.15} C_VEL
LIN {X 0,Y 123.474,Z 453.532,A -85,B 0,C 180,E1 -25906.841,E2 -25906.841} C_VEL
LIN {X 0,Y 128.036,Z 452.327,A -85,B 0,C 180,E1 -25911.089,E2 -25911.089} C_VEL
LIN {X 0,Y 133.938,Z 449.969,A -85,B 0,C 180,E1 -25915.462,E2 -25915.462} C_VEL
LIN {X 0,Y 141.717,Z 445.859,A -85,B 0,C 180,E1 -25920.001,E2 -25920.001} C_VEL
LIN {X 0,Y 147.773,Z 441.94,A -85,B 0,C 180,E1 -25922.991,E2 -25922.991} C_VEL
LIN {X 0,Y 155.499,Z 436.038,A -85,B 0,C 180,E1 -25926.167,E2 -25926.167} C_VEL
LIN {X 0,Y 164.393,Z 427.989,A -85,B 0,C 180,E1 -25929.235,E2 -25929.235} C_VEL
LIN {X 0,Y 172.111,Z 419.648,A -85,B 0,C 180,E1 -25931.503,E2 -25931.503} C_VEL
LIN {X 0,Y 179.959,Z 409.481,A -85,B 0,C 180,E1 -25933.552,E2 -25933.552} C_VEL
LIN {X 0,Y 186.284,Z 399.655,A -85,B 0,C 180,E1 -25935.038,E2 -25935.038} C_VEL
LIN {X 0,Y 192.06,Z 388.851,A -85,B 0,C 180,E1 -25936.287,E2 -25936.287} C_VEL
LIN {X 0,Y 197.751,Z 375.336,A -85,B 0,C 180,E1 -25937.481,E2 -25937.481} C_VEL
LIN {X 0,Y 201.598,Z 363.113,A -85,B 0,C 180,E1 -25938.239,E2 -25938.239} C_VEL
LIN {X 0,Y 204.163,Z 351.626,A -85,B 0,C 180,E1 -25938.765,E2 -25938.765} C_VEL
LIN {X 0,Y 203.752,Z 350.291,A -85,B 0,C 180,E1 -25940.178,E2 -25940.178} C_VEL
LIN {X 0,Y 203.331,Z 349.41,A -85,B 0,C 180,E1 -25942.347,E2 -25942.347} C_VEL
LIN {X 0,Y 203.088,Z 349.763,A -85,B 0,C 180,E1 -25945.604,E2 -25945.604} C_VEL
LIN {X 0,Y 203.147,Z 350.809,A -85,B 0,C 180,E1 -25947.198,E2 -25947.198} C_VEL
LIN {X 0,Y 203.562,Z 354.274,A -85,B 0,C 180,E1 -25950.177,E2 -25950.177} C_VEL
LIN {X 0,Y 203.692,Z 355.185,A -85,B 0,C 180,E1 -25950.765,E2 -25950.765} C_VEL
LIN {X 0,Y 200.253,Z 369.194,A -85,B 0,C 180,E1 -25951.311,E2 -25951.311} C_VEL
LIN {X 0,Y 195.79,Z 382.077,A -85,B 0,C 180,E1 -25952.012,E2 -25952.012} C_VEL
LIN {X 0,Y 190.45,Z 393.914,A -85,B 0,C 180,E1 -25952.92,E2 -25952.92} C_VEL
LIN {X 0,Y 183.65,Z 406.074,A -85,B 0,C 180,E1 -25954.161,E2 -25954.161} C_VEL
LIN {X 0,Y 177.026,Z 415.917,A -85,B 0,C 180,E1 -25955.534,E2 -25955.534} C_VEL
LIN {X 0,Y 169.922,Z 424.911,A -85,B 0,C 180,E1 -25957.241,E2 -25957.241} C_VEL
LIN {X 0,Y 161.72,Z 433.749,A -85,B 0,C 180,E1 -25959.53,E2 -25959.53} C_VEL
LIN {X 0,Y 152.658,Z 442.129,A -85,B 0,C 180,E1 -25962.564,E2 -25962.564} C_VEL
LIN {X 0,Y 145.364,Z 447.896,A -85,B 0,C 180,E1 -25965.495,E2 -25965.495} C_VEL
LIN {X 0,Y 138.587,Z 452.531,A -85,B 0,C 180,E1 -25968.762,E2 -25968.762} C_VEL
LIN {X 0,Y 132.441,Z 456.164,A -85,B 0,C 180,E1 -25972.397,E2 -25972.397} C_VEL
LIN {X 0,Y 127.025,Z 458.919,A -85,B 0,C 180,E1 -25976.412,E2 -25976.412} C_VEL
LIN {X 0,Y 120.9,Z 461.292,A -85,B 0,C 180,E1 -25982.29,E2 -25982.29} C_VEL
LIN {X 0,Y 116.307,Z 462.187,A -85,B 0,C 180,E1 -25988.745,E2 -25988.745} C_VEL
LIN {X 0,Y 113.642,Z 461.653,A -85,B 0,C 180,E1 -25995.679,E2 -25995.679} C_VEL
LIN {X 0,Y 112.632,Z 459.684,A -85,B 0,C 180,E1 -26002.832,E2 -26002.832} C_VEL
LIN {X 0,Y 112.777,Z 456.912,A -85,B 0,C 180,E1 -26008.615,E2 -26008.615} C_VEL
LIN {X 0,Y 112.892,Z 454.84,A -85,B 0,C 180,E1 -26011.783,E2 -26011.783} C_VEL
LIN {X 0,Y 112.875,Z 450.298,A -85,B 0,C 180,E1 -26017.152,E2 -26017.152} C_VEL
LIN {X 0,Y 113.686,Z 443.302,A -85,B 0,C 180,E1 -26023.403,E2 -26023.403} C_VEL
LIN {X 0,Y 115.243,Z 435.662,A -85,B 0,C 180,E1 -26028.67,E2 -26028.67} C_VEL
LIN {X 0,Y 117.193,Z 427.81,A -85,B 0,C 180,E1 -26032.939,E2 -26032.939} C_VEL
LIN {X 0,Y 119.102,Z 420.705,A -85,B 0,C 180,E1 -26036.085,E2 -26036.085} C_VEL
LIN {X 0,Y 119.674,Z 416.192,A -85,B 0,C 180,E1 -26037.901,E2 -26037.901} C_VEL
LIN {X 0,Y 118.906,Z 408.357,A -85,B 0,C 180,E1 -26040.817,E2 -26040.817} C_VEL
LIN {X 0,Y 118.232,Z 400.078,A -85,B 0,C 180,E1 -26043.47,E2 -26043.47} C_VEL
LIN {X 0,Y 118.923,Z 394.864,A -85,B 0,C 180,E1 -26044.792,E2 -26044.792} C_VEL
LIN {X 0,Y 121.736,Z 381.91,A -85,B 0,C 180,E1 -26047.309,E2 -26047.309} C_VEL
LIN {X 0,Y 123.875,Z 369.598,A -85,B 0,C 180,E1 -26049,E2 -26049} C_VEL
LIN {X 0,Y 125.491,Z 356.292,A -85,B 0,C 180,E1 -26050.22,E2 -26050.22} C_VEL
LIN {X 0,Y 128.35,Z 319.386,A -85,B 0,C 180,E1 -26052.644,E2 -26052.644} C_VEL
LIN {X 0,Y 127.107,Z 303.51,A -85,B 0,C 180,E1 -26054.239,E2 -26054.239} C_VEL
LIN {X 0,Y 121.861,Z 286.839,A -85,B 0,C 180,E1 -26057.057,E2 -26057.057} C_VEL
LIN {X 0,Y 116.299,Z 272.27,A -85,B 0,C 180,E1 -26060.052,E2 -26060.052} C_VEL
LIN {X 0,Y 111.082,Z 262.811,A -85,B 0,C 180,E1 -26062.771,E2 -26062.771} C_VEL
LIN {X 0,Y 109.111,Z 259.501,A -85,B 0,C 180,E1 -26063.859,E2 -26063.859} C_VEL
LIN {X 0,Y 107.85,Z 256.904,A -85,B 0,C 180,E1 -26064.632,E2 -26064.632} C_VEL
LIN {X 0,Y 107.692,Z 256.063,A -85,B 0,C 180,E1 -26064.843,E2 -26064.843} C_VEL
LIN {X 0,Y 107.78,Z 256.061,A -85,B 0,C 180,E1 -26068.555,E2 -26068.555} C_VEL
LIN {X 0,Y 107.861,Z 256.047,A -85,B 0,C 180,E1 -26076.985,E2 -26076.985} C_VEL
LIN {X 0,Y 107.954,Z 256.011,A -85,B 0,C 180,E1 -26084.904,E2 -26084.904} C_VEL
LIN {X 0,Y 108.19,Z 256.005,A -85,B 0,C 180,E1 -26088.761,E2 -26088.761} C_VEL
LIN {X 0,Y 108.272,Z 255.996,A -85,B 0,C 180,E1 -26092.539,E2 -26092.539} C_VEL
LIN {X 0,Y 108.864,Z 255.881,A -85,B 0,C 180,E1 -26099.999,E2 -26099.999} C_VEL
LIN {X 0,Y 108.273,Z 255.997,A -85,B 0,C 180,E1 -26107.458,E2 -26107.458} C_VEL
LIN {X 0,Y 108.125,Z 256,A -85,B 0,C 180,E1 -26112.873,E2 -26112.873} C_VEL
LIN {X 0,Y 107.885,Z 255.987,A -85,B 0,C 180,E1 -26119.008,E2 -26119.008} C_VEL
LIN {X 0,Y 107.846,Z 256.033,A -85,B 0,C 180,E1 -26124.184,E2 -26124.184} C_VEL
LIN {X 0,Y 107.778,Z 256.054,A -85,B 0,C 180,E1 -26132.048,E2 -26132.048} C_VEL
LIN {X 0,Y 107.706,Z 256.017,A -85,B 0,C 180,E1 -26138.471,E2 -26138.471} C_VEL
LIN {X 0,Y 107.675,Z 256.063,A -85,B 0,C 180,E1 -26145.886,E2 -26145.886} C_VEL
LIN {X 0,Y 107.681,Z 256.068,A -85,B 0,C 180,E1 -26151.553,E2 -26151.553} C_VEL
LIN {X 0,Y 107.786,Z 256.023,A -85,B 0,C 180,E1 -26158.563,E2 -26158.563} C_VEL
LIN {X 0,Y 107.908,Z 256.041,A -85,B 0,C 180,E1 -26167,E2 -26167} C_VEL
LIN {X 0,Y 108.037,Z 256.025,A -85,B 0,C 180,E1 -26174.92,E2 -26174.92} C_VEL
LIN {X 0,Y 108.285,Z 255.988,A -85,B 0,C 180,E1 -26178.774,E2 -26178.774} C_VEL
LIN {X 0,Y 108.5,Z 256.041,A -85,B 0,C 180,E1 -26186.519,E2 -26186.519} C_VEL
LIN {X 0,Y 109.596,Z 258.898,A -85,B 0,C 180,E1 -26187.243,E2 -26187.243} C_VEL
LIN {X 0,Y 111.353,Z 261.092,A -85,B 0,C 180,E1 -26188.132,E2 -26188.132} C_VEL
LIN {X 0,Y 120.493,Z 279.807,A -85,B 0,C 180,E1 -26192.912,E2 -26192.912} C_VEL
LIN {X 0,Y 127.983,Z 298.249,A -85,B 0,C 180,E1 -26196.51,E2 -26196.51} C_VEL
LIN {X 0,Y 129.351,Z 301.854,A -85,B 0,C 180,E1 -26197.135,E2 -26197.135} C_VEL
LIN {X 0,Y 125.147,Z 350.208,A -85,B 0,C 180,E1 -26200.26,E2 -26200.26} C_VEL
LIN {X 0,Y 123.519,Z 363.242,A -85,B 0,C 180,E1 -26201.694,E2 -26201.694} C_VEL
LIN {X 0,Y 121.191,Z 376.702,A -85,B 0,C 180,E1 -26203.839,E2 -26203.839} C_VEL
LIN {X 0,Y 118.17,Z 390.094,A -85,B 0,C 180,E1 -26206.8,E2 -26206.8} C_VEL
LIN {X 0,Y 115.465,Z 400.953,A -85,B 0,C 180,E1 -26210.02,E2 -26210.02} C_VEL
LIN {X 0,Y 112.577,Z 411.474,A -85,B 0,C 180,E1 -26214.042,E2 -26214.042} C_VEL
LIN {X 0,Y 109.701,Z 421.56,A -85,B 0,C 180,E1 -26219.03,E2 -26219.03} C_VEL
LIN {X 0,Y 107.55,Z 429.582,A -85,B 0,C 180,E1 -26224.169,E2 -26224.169} C_VEL
LIN {X 0,Y 106.068,Z 436.57,A -85,B 0,C 180,E1 -26229.847,E2 -26229.847} C_VEL
LIN {X 0,Y 105.182,Z 441.887,A -85,B 0,C 180,E1 -26235.315,E2 -26235.315} C_VEL
LIN {X 0,Y 104.971,Z 447.502,A -85,B 0,C 180,E1 -26242.948,E2 -26242.948} C_VEL
LIN {X 0,Y 106.075,Z 450.887,A -85,B 0,C 180,E1 -26249.455,E2 -26249.455} C_VEL
LIN {X 0,Y 109.037,Z 453.459,A -85,B 0,C 180,E1 -26257.25,E2 -26257.25} C_VEL
LIN {X 0,Y 111.655,Z 454.164,A -85,B 0,C 180,E1 -26261.657,E2 -26261.657} C_VEL
LIN {X 0,Y 115.555,Z 454.265,A -85,B 0,C 180,E1 -26266.659,E2 -26266.659} C_VEL
LIN {X 0,Y 120.73,Z 453.401,A -85,B 0,C 180,E1 -26271.692,E2 -26271.692} C_VEL
LIN {X 0,Y 127.594,Z 451.2,A -85,B 0,C 180,E1 -26276.844,E2 -26276.844} C_VEL
LIN {X 0,Y 135.997,Z 447.378,A -85,B 0,C 180,E1 -26281.65,E2 -26281.65} C_VEL
LIN {X 0,Y 144.409,Z 442.383,A -85,B 0,C 180,E1 -26285.587,E2 -26285.587} C_VEL
LIN {X 0,Y 152.409,Z 436.668,A -85,B 0,C 180,E1 -26288.621,E2 -26288.621} C_VEL
LIN {X 0,Y 160.866,Z 429.456,A -85,B 0,C 180,E1 -26291.339,E2 -26291.339} C_VEL
LIN {X 0,Y 168.578,Z 421.66,A -85,B 0,C 180,E1 -26293.478,E2 -26293.478} C_VEL
LIN {X 0,Y 176.731,Z 411.888,A -85,B 0,C 180,E1 -26295.464,E2 -26295.464} C_VEL
LIN {X 0,Y 183.694,Z 401.835,A -85,B 0,C 180,E1 -26296.986,E2 -26296.986} C_VEL
LIN {X 0,Y 189.314,Z 392.09,A -85,B 0,C 180,E1 -26298.116,E2 -26298.116} C_VEL
LIN {X 0,Y 194.971,Z 379.986,A -85,B 0,C 180,E1 -26299.206,E2 -26299.206} C_VEL
LIN {X 0,Y 199.249,Z 367.965,A -85,B 0,C 180,E1 -26300.015,E2 -26300.015} C_VEL
LIN {X 0,Y 202.152,Z 357.094,A -85,B 0,C 180,E1 -26300.552,E2 -26300.552} C_VEL
LIN {X 0,Y 201.874,Z 356.351,A -85,B 0,C 180,E1 -26302.517,E2 -26302.517} C_VEL
LIN {X 0,Y 201.663,Z 356.711,A -85,B 0,C 180,E1 -26305.507,E2 -26305.507} C_VEL
LIN {X 0,Y 201.634,Z 357.928,A -85,B 0,C 180,E1 -26307.078,E2 -26307.078} C_VEL
LIN {X 0,Y 201.71,Z 359.845,A -85,B 0,C 180,E1 -26308.893,E2 -26308.893} C_VEL
LIN {X 0,Y 198.882,Z 370.203,A -85,B 0,C 180,E1 -26309.329,E2 -26309.329} C_VEL
LIN {X 0,Y 194.626,Z 382.017,A -85,B 0,C 180,E1 -26309.94,E2 -26309.94} C_VEL
LIN {X 0,Y 189.146,Z 393.805,A -85,B 0,C 180,E1 -26310.778,E2 -26310.778} C_VEL
LIN {X 0,Y 182.169,Z 405.84,A -85,B 0,C 180,E1 -26311.934,E2 -26311.934} C_VEL
LIN {X 0,Y 174.593,Z 416.546,A -85,B 0,C 180,E1 -26313.366,E2 -26313.366} C_VEL
LIN {X 0,Y 165.824,Z 426.917,A -85,B 0,C 180,E1 -26315.336,E2 -26315.336} C_VEL
LIN {X 0,Y 157.395,Z 435.374,A -85,B 0,C 180,E1 -26317.581,E2 -26317.581} C_VEL
LIN {X 0,Y 149.309,Z 442.263,A -85,B 0,C 180,E1 -26320.11,E2 -26320.11} C_VEL
LIN {X 0,Y 140.424,Z 448.697,A -85,B 0,C 180,E1 -26323.479,E2 -26323.479} C_VEL
LIN {X 0,Y 133.359,Z 453.099,A -85,B 0,C 180,E1 -26326.762,E2 -26326.762} C_VEL
LIN {X 0,Y 128.968,Z 455.476,A -85,B 0,C 180,E1 -26329.167,E2 -26329.167} C_VEL
LIN {X 0,Y 121.157,Z 459.065,A -85,B 0,C 180,E1 -26334.548,E2 -26334.548} C_VEL
LIN {X 0,Y 114.647,Z 461.144,A -85,B 0,C 180,E1 -26340.636,E2 -26340.636} C_VEL
LIN {X 0,Y 109.71,Z 461.798,A -85,B 0,C 180,E1 -26347.398,E2 -26347.398} C_VEL
LIN {X 0,Y 106.756,Z 461.074,A -85,B 0,C 180,E1 -26354.734,E2 -26354.734} C_VEL
LIN {X 0,Y 105.634,Z 458.834,A -85,B 0,C 180,E1 -26362.354,E2 -26362.354} C_VEL
LIN {X 0,Y 105.789,Z 455.774,A -85,B 0,C 180,E1 -26368.684,E2 -26368.684} C_VEL
LIN {X 0,Y 105.837,Z 453.042,A -85,B 0,C 180,E1 -26372.78,E2 -26372.78} C_VEL
LIN {X 0,Y 105.864,Z 448.937,A -85,B 0,C 180,E1 -26377.629,E2 -26377.629} C_VEL
LIN {X 0,Y 106.611,Z 442.857,A -85,B 0,C 180,E1 -26383.338,E2 -26383.338} C_VEL
LIN {X 0,Y 108.174,Z 435.185,A -85,B 0,C 180,E1 -26388.954,E2 -26388.954} C_VEL
LIN {X 0,Y 110.2,Z 427.3,A -85,B 0,C 180,E1 -26393.487,E2 -26393.487} C_VEL
LIN {X 0,Y 113.201,Z 416.631,A -85,B 0,C 180,E1 -26398.251,E2 -26398.251} C_VEL
LIN {X 0,Y 116.062,Z 406.203,A -85,B 0,C 180,E1 -26401.832,E2 -26401.832} C_VEL
LIN {X 0,Y 118.923,Z 394.864,A -85,B 0,C 180,E1 -26404.792,E2 -26404.792} C_VEL
LIN {X 0,Y 119.625,Z 389.609,A -85,B 0,C 180,E1 -26405.999,E2 -26405.999} C_VEL
LIN {X 0,Y 119.371,Z 384.234,A -85,B 0,C 180,E1 -26407.251,E2 -26407.251} C_VEL
LIN {X 0,Y 117.76,Z 371.531,A -85,B 0,C 180,E1 -26409.931,E2 -26409.931} C_VEL
LIN {X 0,Y 117.914,Z 365.846,A -85,B 0,C 180,E1 -26410.749,E2 -26410.749} C_VEL
LIN {X 0,Y 119.414,Z 351.799,A -85,B 0,C 180,E1 -26411.937,E2 -26411.937} C_VEL
LIN {X 0,Y 122.006,Z 319.563,A -85,B 0,C 180,E1 -26414.128,E2 -26414.128} C_VEL
LIN {X 0,Y 120.905,Z 305.313,A -85,B 0,C 180,E1 -26415.668,E2 -26415.668} C_VEL
LIN {X 0,Y 115.581,Z 288.192,A -85,B 0,C 180,E1 -26418.747,E2 -26418.747} C_VEL
LIN {X 0,Y 110.574,Z 275.308,A -85,B 0,C 180,E1 -26421.663,E2 -26421.663} C_VEL
LIN {X 0,Y 104.709,Z 264.558,A -85,B 0,C 180,E1 -26425.066,E2 -26425.066} C_VEL
LIN {X 0,Y 102.164,Z 260.438,A -85,B 0,C 180,E1 -26426.609,E2 -26426.609} C_VEL
LIN {X 0,Y 100.919,Z 257.982,A -85,B 0,C 180,E1 -26427.457,E2 -26427.457} C_VEL
LIN {X 0,Y 100.724,Z 256.935,A -85,B 0,C 180,E1 -26427.689,E2 -26427.689} C_VEL
LIN {X 0,Y 100.734,Z 256.926,A -85,B 0,C 180,E1 -26435.252,E2 -26435.252} C_VEL
LIN {X 0,Y 100.765,Z 256.931,A -85,B 0,C 180,E1 -26439.589,E2 -26439.589} C_VEL
LIN {X 0,Y 101.1,Z 256.884,A -85,B 0,C 180,E1 -26447.961,E2 -26447.961} C_VEL
LIN {X 0,Y 101.206,Z 256.877,A -85,B 0,C 180,E1 -26452.015,E2 -26452.015} C_VEL
LIN {X 0,Y 101.795,Z 256.76,A -85,B 0,C 180,E1 -26459.999,E2 -26459.999} C_VEL
LIN {X 0,Y 101.21,Z 256.877,A -85,B 0,C 180,E1 -26467.982,E2 -26467.982} C_VEL
LIN {X 0,Y 101.061,Z 256.875,A -85,B 0,C 180,E1 -26473.226,E2 -26473.226} C_VEL
LIN {X 0,Y 100.8,Z 256.873,A -85,B 0,C 180,E1 -26480.401,E2 -26480.401} C_VEL
LIN {X 0,Y 100.764,Z 256.918,A -85,B 0,C 180,E1 -26484.96,E2 -26484.96} C_VEL
LIN {X 0,Y 100.687,Z 256.932,A -85,B 0,C 180,E1 -26493.123,E2 -26493.123} C_VEL
LIN {X 0,Y 100.654,Z 256.891,A -85,B 0,C 180,E1 -26499.829,E2 -26499.829} C_VEL
LIN {X 0,Y 100.647,Z 256.938,A -85,B 0,C 180,E1 -26505.717,E2 -26505.717} C_VEL
LIN {X 0,Y 100.62,Z 256.95,A -85,B 0,C 180,E1 -26511.057,E2 -26511.057} C_VEL
LIN {X 0,Y 100.682,Z 256.905,A -85,B 0,C 180,E1 -26516.89,E2 -26516.89} C_VEL
LIN {X 0,Y 100.782,Z 256.933,A -85,B 0,C 180,E1 -26525.269,E2 -26525.269} C_VEL
LIN {X 0,Y 100.815,Z 256.908,A -85,B 0,C 180,E1 -26529.604,E2 -26529.604} C_VEL
LIN {X 0,Y 101.185,Z 256.878,A -85,B 0,C 180,E1 -26537.975,E2 -26537.975} C_VEL
LIN {X 0,Y 101.271,Z 256.871,A -85,B 0,C 180,E1 -26543.526,E2 -26543.526} C_VEL
LIN {X 0,Y 102.331,Z 259.745,A -85,B 0,C 180,E1 -26544.387,E2 -26544.387} C_VEL
LIN {X 0,Y 104.098,Z 262.116,A -85,B 0,C 180,E1 -26545.414,E2 -26545.414} C_VEL
LIN {X 0,Y 107.465,Z 267.437,A -85,B 0,C 180,E1 -26547.329,E2 -26547.329} C_VEL
LIN {X 0,Y 115.306,Z 284.14,A -85,B 0,C 180,E1 -26551.771,E2 -26551.771} C_VEL
LIN {X 0,Y 122.172,Z 301.317,A -85,B 0,C 180,E1 -26555.284,E2 -26555.284} C_VEL
LIN {X 0,Y 122.969,Z 303.441,A -85,B 0,C 180,E1 -26555.682,E2 -26555.682} C_VEL
LIN {X 0,Y 118.739,Z 350.259,A -85,B 0,C 180,E1 -26558.829,E2 -26558.829} C_VEL
LIN {X 0,Y 116.965,Z 363.763,A -85,B 0,C 180,E1 -26560.384,E2 -26560.384} C_VEL
LIN {X 0,Y 114.674,Z 376.434,A -85,B 0,C 180,E1 -26562.486,E2 -26562.486} C_VEL
LIN {X 0,Y 111.657,Z 389.316,A -85,B 0,C 180,E1 -26565.436,E2 -26565.436} C_VEL
LIN {X 0,Y 108.777,Z 400.47,A -85,B 0,C 180,E1 -26568.845,E2 -26568.845} C_VEL
LIN {X 0,Y 105.945,Z 410.373,A -85,B 0,C 180,E1 -26572.761,E2 -26572.761} C_VEL
LIN {X 0,Y 103.111,Z 419.965,A -85,B 0,C 180,E1 -26577.619,E2 -26577.619} C_VEL
LIN {X 0,Y 100.714,Z 428.486,A -85,B 0,C 180,E1 -26583.138,E2 -26583.138} C_VEL
LIN {X 0,Y 99.184,Z 435.342,A -85,B 0,C 180,E1 -26588.793,E2 -26588.793} C_VEL
LIN {X 0,Y 98.024,Z 441.909,A -85,B 0,C 180,E1 -26595.798,E2 -26595.798} C_VEL
LIN {X 0,Y 97.855,Z 446.489,A -85,B 0,C 180,E1 -26602.18,E2 -26602.18} C_VEL
LIN {X 0,Y 99.127,Z 450.771,A -85,B 0,C 180,E1 -26610.247,E2 -26610.247} C_VEL
LIN {X 0,Y 100.8,Z 452.636,A -85,B 0,C 180,E1 -26615.272,E2 -26615.272} C_VEL
LIN {X 0,Y 103.899,Z 454.13,A -85,B 0,C 180,E1 -26621.243,E2 -26621.243} C_VEL
LIN {X 0,Y 108.158,Z 454.702,A -85,B 0,C 180,E1 -26627.053,E2 -26627.053} C_VEL
LIN {X 0,Y 114.04,Z 454.181,A -85,B 0,C 180,E1 -26632.921,E2 -26632.921} C_VEL
LIN {X 0,Y 119.608,Z 452.886,A -85,B 0,C 180,E1 -26637.185,E2 -26637.185} C_VEL
LIN {X 0,Y 126.531,Z 450.469,A -85,B 0,C 180,E1 -26641.441,E2 -26641.441} C_VEL
LIN {X 0,Y 135.707,Z 446.159,A -85,B 0,C 180,E1 -26645.946,E2 -26645.946} C_VEL
LIN {X 0,Y 145.432,Z 440.294,A -85,B 0,C 180,E1 -26649.76,E2 -26649.76} C_VEL
LIN {X 0,Y 154.503,Z 433.512,A -85,B 0,C 180,E1 -26652.654,E2 -26652.654} C_VEL
